LIN {X 0,Y 401.236,Z 607.436,A -85,B 0,C 180,E1 -18756.409,E2 -18756.409} C_VEL
LIN {X 0,Y 401.176,Z 607.446,A -85,B 0,C 180,E1 -18759.805,E2 -18759.805} C_VEL
LIN {X 0,Y 401.178,Z 607.441,A -85,B 0,C 180,E1 -18762.916,E2 -18762.916} C_VEL
LIN {X 0,Y 401.243,Z 607.437,A -85,B 0,C 180,E1 -18765.711,E2 -18765.711} C_VEL
LIN {X 0,Y 401.184,Z 607.441,A -85,B 0,C 180,E1 -18768.656,E2 -18768.656} C_VEL
LIN {X 0,Y 401.211,Z 607.44,A -85,B 0,C 180,E1 -18772.335,E2 -18772.335} C_VEL
LIN {X 0,Y 401.205,Z 607.445,A -85,B 0,C 180,E1 -18776.036,E2 -18776.036} C_VEL
LIN {X 0,Y 401.214,Z 607.439,A -85,B 0,C 180,E1 -18779.583,E2 -18779.583} C_VEL
LIN {X 0,Y 401.241,Z 607.433,A -85,B 0,C 180,E1 -18783.007,E2 -18783.007} C_VEL
LIN {X 0,Y 401.328,Z 607.551,A -85,B 0,C 180,E1 -18783.748,E2 -18783.748} C_VEL
LIN {X 0,Y 403.625,Z 620.57,A -85,B 0,C 180,E1 -18786.89,E2 -18786.89} C_VEL
LIN {X 0,Y 403.581,Z 624.602,A -85,B 0,C 180,E1 -18787.822,E2 -18787.822} C_VEL
LIN {X 0,Y 402.02,Z 640.648,A -85,B 0,C 180,E1 -18791.46,E2 -18791.46} C_VEL
LIN {X 0,Y 401.655,Z 644.543,A -85,B 0,C 180,E1 -18792.313,E2 -18792.313} C_VEL
LIN {X 0,Y 404.651,Z 676.358,A -85,B 0,C 180,E1 -18793.161,E2 -18793.161} C_VEL
LIN {X 0,Y 405.065,Z 683.005,A -85,B 0,C 180,E1 -18793.331,E2 -18793.331} C_VEL
LIN {X 0,Y 403.56,Z 750.603,A -85,B 0,C 180,E1 -18794.942,E2 -18794.942} C_VEL
LIN {X 0,Y 403.184,Z 761.472,A -85,B 0,C 180,E1 -18795.313,E2 -18795.313} C_VEL
LIN {X 0,Y 402.795,Z 771.537,A -85,B 0,C 180,E1 -18795.781,E2 -18795.781} C_VEL
LIN {X 0,Y 402.347,Z 782.009,A -85,B 0,C 180,E1 -18796.407,E2 -18796.407} C_VEL
LIN {X 0,Y 401.883,Z 790.591,A -85,B 0,C 180,E1 -18797.033,E2 -18797.033} C_VEL
LIN {X 0,Y 401.239,Z 800.472,A -85,B 0,C 180,E1 -18797.908,E2 -18797.908} C_VEL
LIN {X 0,Y 400.952,Z 807.903,A -85,B 0,C 180,E1 -18798.679,E2 -18798.679} C_VEL
LIN {X 0,Y 400.256,Z 817.734,A -85,B 0,C 180,E1 -18799.922,E2 -18799.922} C_VEL
LIN {X 0,Y 399.876,Z 824.495,A -85,B 0,C 180,E1 -18800.93,E2 -18800.93} C_VEL
LIN {X 0,Y 399.455,Z 831.571,A -85,B 0,C 180,E1 -18802.19,E2 -18802.19} C_VEL
LIN {X 0,Y 399.275,Z 837.486,A -85,B 0,C 180,E1 -18803.453,E2 -18803.453} C_VEL
LIN {X 0,Y 399.089,Z 843.17,A -85,B 0,C 180,E1 -18804.966,E2 -18804.966} C_VEL
LIN {X 0,Y 399.008,Z 847.589,A -85,B 0,C 180,E1 -18806.478,E2 -18806.478} C_VEL
LIN {X 0,Y 398.99,Z 850.871,A -85,B 0,C 180,E1 -18807.988,E2 -18807.988} C_VEL
LIN {X 0,Y 398.984,Z 852.53,A -85,B 0,C 180,E1 -18808.994,E2 -18808.994} C_VEL
LIN {X 0,Y 398.913,Z 854.339,A -85,B 0,C 180,E1 -18811.006,E2 -18811.006} C_VEL
LIN {X 0,Y 398.916,Z 854.625,A -85,B 0,C 180,E1 -18812.013,E2 -18812.013} C_VEL
LIN {X 0,Y 398.936,Z 853.919,A -85,B 0,C 180,E1 -18814.027,E2 -18814.027} C_VEL
LIN {X 0,Y 399.279,Z 851.395,A -85,B 0,C 180,E1 -18816.042,E2 -18816.042} C_VEL
LIN {X 0,Y 399.537,Z 849.602,A -85,B 0,C 180,E1 -18817.049,E2 -18817.049} C_VEL
LIN {X 0,Y 400.122,Z 845.914,A -85,B 0,C 180,E1 -18818.558,E2 -18818.558} C_VEL
LIN {X 0,Y 400.877,Z 841.119,A -85,B 0,C 180,E1 -18820.063,E2 -18820.063} C_VEL
LIN {X 0,Y 402.106,Z 835.034,A -85,B 0,C 180,E1 -18821.556,E2 -18821.556} C_VEL
LIN {X 0,Y 403.485,Z 827.462,A -85,B 0,C 180,E1 -18823.043,E2 -18823.043} C_VEL
LIN {X 0,Y 404.619,Z 820.376,A -85,B 0,C 180,E1 -18824.204,E2 -18824.204} C_VEL
LIN {X 0,Y 406.142,Z 811.671,A -85,B 0,C 180,E1 -18825.377,E2 -18825.377} C_VEL
LIN {X 0,Y 407.485,Z 803.092,A -85,B 0,C 180,E1 -18826.349,E2 -18826.349} C_VEL
LIN {X 0,Y 408.792,Z 794.302,A -85,B 0,C 180,E1 -18827.192,E2 -18827.192} C_VEL
LIN {X 0,Y 410.234,Z 783.638,A -85,B 0,C 180,E1 -18828.028,E2 -18828.028} C_VEL
LIN {X 0,Y 411.505,Z 773.302,A -85,B 0,C 180,E1 -18828.676,E2 -18828.676} C_VEL
LIN {X 0,Y 412.645,Z 762.627,A -85,B 0,C 180,E1 -18829.201,E2 -18829.201} C_VEL
LIN {X 0,Y 413.498,Z 751.718,A -85,B 0,C 180,E1 -18829.61,E2 -18829.61} C_VEL
LIN {X 0,Y 415.326,Z 717.984,A -85,B 0,C 180,E1 -18830.484,E2 -18830.484} C_VEL
LIN {X 0,Y 416.908,Z 685.447,A -85,B 0,C 180,E1 -18831.33,E2 -18831.33} C_VEL
LIN {X 0,Y 415.184,Z 672.854,A -85,B 0,C 180,E1 -18831.892,E2 -18831.892} C_VEL
LIN {X 0,Y 411.389,Z 654.895,A -85,B 0,C 180,E1 -18832.847,E2 -18832.847} C_VEL
LIN {X 0,Y 407.995,Z 642.009,A -85,B 0,C 180,E1 -18833.66,E2 -18833.66} C_VEL
LIN {X 0,Y 408.232,Z 638.669,A -85,B 0,C 180,E1 -18834.581,E2 -18834.581} C_VEL
LIN {X 0,Y 406.942,Z 630.553,A -85,B 0,C 180,E1 -18837.137,E2 -18837.137} C_VEL
LIN {X 0,Y 405.56,Z 623.765,A -85,B 0,C 180,E1 -18839.487,E2 -18839.487} C_VEL
LIN {X 0,Y 404.026,Z 617.69,A -85,B 0,C 180,E1 -18841.843,E2 -18841.843} C_VEL
LIN {X 0,Y 402.495,Z 611.781,A -85,B 0,C 180,E1 -18844.417,E2 -18844.417} C_VEL
LIN {X 0,Y 401.245,Z 607.433,A -85,B 0,C 180,E1 -18846.636,E2 -18846.636} C_VEL
LIN {X 0,Y 401.201,Z 607.432,A -85,B 0,C 180,E1 -18849.809,E2 -18849.809} C_VEL
LIN {X 0,Y 401.216,Z 607.436,A -85,B 0,C 180,E1 -18852.912,E2 -18852.912} C_VEL
LIN {X 0,Y 401.249,Z 607.434,A -85,B 0,C 180,E1 -18855.712,E2 -18855.712} C_VEL
LIN {X 0,Y 401.218,Z 607.439,A -85,B 0,C 180,E1 -18858.651,E2 -18858.651} C_VEL
LIN {X 0,Y 401.253,Z 607.437,A -85,B 0,C 180,E1 -18861.771,E2 -18861.771} C_VEL
LIN {X 0,Y 401.255,Z 607.436,A -85,B 0,C 180,E1 -18865.13,E2 -18865.13} C_VEL
LIN {X 0,Y 401.243,Z 607.439,A -85,B 0,C 180,E1 -18868.803,E2 -18868.803} C_VEL
LIN {X 0,Y 401.259,Z 607.435,A -85,B 0,C 180,E1 -18871.88,E2 -18871.88} C_VEL
LIN {X 0,Y 401.272,Z 607.436,A -85,B 0,C 180,E1 -18875.232,E2 -18875.232} C_VEL
LIN {X 0,Y 401.283,Z 607.543,A -85,B 0,C 180,E1 -18876.603,E2 -18876.603} C_VEL
LIN {X 0,Y 403.001,Z 613.819,A -85,B 0,C 180,E1 -18879.811,E2 -18879.811} C_VEL
LIN {X 0,Y 404.416,Z 619.422,A -85,B 0,C 180,E1 -18882.288,E2 -18882.288} C_VEL
LIN {X 0,Y 406.124,Z 627.38,A -85,B 0,C 180,E1 -18885.409,E2 -18885.409} C_VEL
LIN {X 0,Y 406.574,Z 629.868,A -85,B 0,C 180,E1 -18886.249,E2 -18886.249} C_VEL
LIN {X 0,Y 412.813,Z 642.686,A -85,B 0,C 180,E1 -18887.379,E2 -18887.379} C_VEL
LIN {X 0,Y 414.891,Z 649.227,A -85,B 0,C 180,E1 -18887.801,E2 -18887.801} C_VEL
LIN {X 0,Y 417.902,Z 663.56,A -85,B 0,C 180,E1 -18888.553,E2 -18888.553} C_VEL
LIN {X 0,Y 414.716,Z 719.256,A -85,B 0,C 180,E1 -18889.969,E2 -18889.969} C_VEL
LIN {X 0,Y 413.649,Z 739.357,A -85,B 0,C 180,E1 -18890.527,E2 -18890.527} C_VEL
LIN {X 0,Y 412.557,Z 752.584,A -85,B 0,C 180,E1 -18891.087,E2 -18891.087} C_VEL
LIN {X 0,Y 411.542,Z 762.975,A -85,B 0,C 180,E1 -18891.682,E2 -18891.682} C_VEL
LIN {X 0,Y 410.218,Z 774.378,A -85,B 0,C 180,E1 -18892.515,E2 -18892.515} C_VEL
LIN {X 0,Y 409.038,Z 783.376,A -85,B 0,C 180,E1 -18893.318,E2 -18893.318} C_VEL
LIN {X 0,Y 407.647,Z 792.758,A -85,B 0,C 180,E1 -18894.33,E2 -18894.33} C_VEL
LIN {X 0,Y 406.417,Z 800.413,A -85,B 0,C 180,E1 -18895.304,E2 -18895.304} C_VEL
LIN {X 0,Y 404.921,Z 808.487,A -85,B 0,C 180,E1 -18896.529,E2 -18896.529} C_VEL
LIN {X 0,Y 403.576,Z 815.234,A -85,B 0,C 180,E1 -18897.762,E2 -18897.762} C_VEL
LIN {X 0,Y 402.452,Z 820.862,A -85,B 0,C 180,E1 -18899.002,E2 -18899.002} C_VEL
LIN {X 0,Y 401.386,Z 826.302,A -85,B 0,C 180,E1 -18900.5,E2 -18900.5} C_VEL
LIN {X 0,Y 400.433,Z 830.57,A -85,B 0,C 180,E1 -18902.005,E2 -18902.005} C_VEL
LIN {X 0,Y 399.986,Z 833.639,A -85,B 0,C 180,E1 -18903.464,E2 -18903.464} C_VEL
LIN {X 0,Y 399.34,Z 836.196,A -85,B 0,C 180,E1 -18905.342,E2 -18905.342} C_VEL
LIN {X 0,Y 399.176,Z 836.861,A -85,B 0,C 180,E1 -18906.043,E2 -18906.043} C_VEL
LIN {X 0,Y 398.808,Z 837.317,A -85,B 0,C 180,E1 -18908.077,E2 -18908.077} C_VEL
LIN {X 0,Y 398.775,Z 836.922,A -85,B 0,C 180,E1 -18909.095,E2 -18909.095} C_VEL
LIN {X 0,Y 398.83,Z 835.693,A -85,B 0,C 180,E1 -18910.421,E2 -18910.421} C_VEL
LIN {X 0,Y 398.746,Z 833,A -85,B 0,C 180,E1 -18912.168,E2 -18912.168} C_VEL
LIN {X 0,Y 398.994,Z 827.975,A -85,B 0,C 180,E1 -18914.227,E2 -18914.227} C_VEL
LIN {X 0,Y 399.221,Z 822.72,A -85,B 0,C 180,E1 -18915.78,E2 -18915.78} C_VEL
LIN {X 0,Y 399.477,Z 817.276,A -85,B 0,C 180,E1 -18917.079,E2 -18917.079} C_VEL
LIN {X 0,Y 399.836,Z 810.653,A -85,B 0,C 180,E1 -18918.38,E2 -18918.38} C_VEL
LIN {X 0,Y 400.296,Z 802.586,A -85,B 0,C 180,E1 -18919.684,E2 -18919.684} C_VEL
LIN {X 0,Y 400.729,Z 794.881,A -85,B 0,C 180,E1 -18920.729,E2 -18920.729} C_VEL
LIN {X 0,Y 401.198,Z 785.777,A -85,B 0,C 180,E1 -18921.764,E2 -18921.764} C_VEL
LIN {X 0,Y 401.706,Z 777.528,A -85,B 0,C 180,E1 -18922.557,E2 -18922.557} C_VEL
LIN {X 0,Y 402.234,Z 767.766,A -85,B 0,C 180,E1 -18923.338,E2 -18923.338} C_VEL
LIN {X 0,Y 402.762,Z 756.608,A -85,B 0,C 180,E1 -18924.054,E2 -18924.054} C_VEL
LIN {X 0,Y 403.039,Z 746.109,A -85,B 0,C 180,E1 -18924.583,E2 -18924.583} C_VEL
LIN {X 0,Y 403.458,Z 734.818,A -85,B 0,C 180,E1 -18925,E2 -18925} C_VEL
LIN {X 0,Y 404.11,Z 711.349,A -85,B 0,C 180,E1 -18925.58,E2 -18925.58} C_VEL
LIN {X 0,Y 405.406,Z 654.841,A -85,B 0,C 180,E1 -18926.917,E2 -18926.917} C_VEL
LIN {X 0,Y 402.416,Z 630.593,A -85,B 0,C 180,E1 -18927.582,E2 -18927.582} C_VEL
LIN {X 0,Y 402.044,Z 626.481,A -85,B 0,C 180,E1 -18927.712,E2 -18927.712} C_VEL
LIN {X 0,Y 402.802,Z 616.204,A -85,B 0,C 180,E1 -18930.284,E2 -18930.284} C_VEL
LIN {X 0,Y 401.358,Z 607.42,A -85,B 0,C 180,E1 -18932.603,E2 -18932.603} C_VEL
LIN {X 0,Y 401.245,Z 607.435,A -85,B 0,C 180,E1 -18936.407,E2 -18936.407} C_VEL
LIN {X 0,Y 401.219,Z 607.441,A -85,B 0,C 180,E1 -18939.812,E2 -18939.812} C_VEL
LIN {X 0,Y 401.232,Z 607.434,A -85,B 0,C 180,E1 -18942.908,E2 -18942.908} C_VEL
LIN {X 0,Y 401.276,Z 607.433,A -85,B 0,C 180,E1 -18945.716,E2 -18945.716} C_VEL
LIN {X 0,Y 401.209,Z 607.438,A -85,B 0,C 180,E1 -18948.651,E2 -18948.651} C_VEL
LIN {X 0,Y 401.249,Z 607.437,A -85,B 0,C 180,E1 -18951.77,E2 -18951.77} C_VEL
LIN {X 0,Y 401.253,Z 607.432,A -85,B 0,C 180,E1 -18955.129,E2 -18955.129} C_VEL
LIN {X 0,Y 401.237,Z 607.434,A -85,B 0,C 180,E1 -18958.803,E2 -18958.803} C_VEL
LIN {X 0,Y 401.254,Z 607.437,A -85,B 0,C 180,E1 -18961.88,E2 -18961.88} C_VEL
LIN {X 0,Y 401.266,Z 607.43,A -85,B 0,C 180,E1 -18965.232,E2 -18965.232} C_VEL
LIN {X 0,Y 401.249,Z 607.434,A -85,B 0,C 180,E1 -18968.494,E2 -18968.494} C_VEL
LIN {X 0,Y 401.293,Z 607.43,A -85,B 0,C 180,E1 -18971.688,E2 -18971.688} C_VEL
LIN {X 0,Y 401.332,Z 607.422,A -85,B 0,C 180,E1 -18974.823,E2 -18974.823} C_VEL
LIN {X 0,Y 401.433,Z 607.416,A -85,B 0,C 180,E1 -18977.914,E2 -18977.914} C_VEL
LIN {X 0,Y 401.48,Z 607.411,A -85,B 0,C 180,E1 -18981.977,E2 -18981.977} C_VEL
LIN {X 0,Y 401.588,Z 607.39,A -85,B 0,C 180,E1 -18984.997,E2 -18984.997} C_VEL
LIN {X 0,Y 401.466,Z 607.412,A -85,B 0,C 180,E1 -18988,E2 -18988} C_VEL
LIN {X 0,Y 401.576,Z 607.399,A -85,B 0,C 180,E1 -18990,E2 -18990} C_VEL
LIN {X 0,Y 401.579,Z 607.398,A -85,B 0,C 180,E1 -18994.001,E2 -18994.001} C_VEL
LIN {X 0,Y 401.5,Z 607.401,A -85,B 0,C 180,E1 -18997.014,E2 -18997.014} C_VEL
LIN {X 0,Y 401.374,Z 607.423,A -85,B 0,C 180,E1 -19000.05,E2 -19000.05} C_VEL
LIN {X 0,Y 401.371,Z 607.417,A -85,B 0,C 180,E1 -19003.113,E2 -19003.113} C_VEL
LIN {X 0,Y 401.354,Z 607.423,A -85,B 0,C 180,E1 -19006.291,E2 -19006.291} C_VEL
LIN {X 0,Y 401.313,Z 607.426,A -85,B 0,C 180,E1 -19009.525,E2 -19009.525} C_VEL
LIN {X 0,Y 401.267,Z 607.431,A -85,B 0,C 180,E1 -19012.583,E2 -19012.583} C_VEL
LIN {X 0,Y 401.279,Z 607.434,A -85,B 0,C 180,E1 -19015.873,E2 -19015.873} C_VEL
LIN {X 0,Y 401.264,Z 607.431,A -85,B 0,C 180,E1 -19019.259,E2 -19019.259} C_VEL
LIN {X 0,Y 401.269,Z 607.43,A -85,B 0,C 180,E1 -19022.76,E2 -19022.76} C_VEL
LIN {X 0,Y 401.311,Z 607.427,A -85,B 0,C 180,E1 -19026.401,E2 -19026.401} C_VEL
LIN {X 0,Y 401.274,Z 607.429,A -85,B 0,C 180,E1 -19028.932,E2 -19028.932} C_VEL
LIN {X 0,Y 401.23,Z 607.435,A -85,B 0,C 180,E1 -19032.909,E2 -19032.909} C_VEL
LIN {X 0,Y 401.274,Z 607.433,A -85,B 0,C 180,E1 -19035.716,E2 -19035.716} C_VEL
LIN {X 0,Y 401.234,Z 607.438,A -85,B 0,C 180,E1 -19039.766,E2 -19039.766} C_VEL
LIN {X 0,Y 401.256,Z 607.434,A -85,B 0,C 180,E1 -19042.341,E2 -19042.341} C_VEL
LIN {X 0,Y 401.258,Z 607.431,A -85,B 0,C 180,E1 -19045.129,E2 -19045.129} C_VEL
LIN {X 0,Y 401.238,Z 607.434,A -85,B 0,C 180,E1 -19048.803,E2 -19048.803} C_VEL
LIN {X 0,Y 401.255,Z 607.437,A -85,B 0,C 180,E1 -19051.88,E2 -19051.88} C_VEL
LIN {X 0,Y 401.257,Z 607.431,A -85,B 0,C 180,E1 -19055.144,E2 -19055.144} C_VEL
LIN {X 0,Y 400.613,Z 607.519,A -85,B 0,C 180,E1 -19055.982,E2 -19055.982} C_VEL
LIN {X 0,Y 397.749,Z 607.869,A -85,B 0,C 180,E1 -19057.345,E2 -19057.345} C_VEL
LIN {X 0,Y 395.32,Z 608.173,A -85,B 0,C 180,E1 -19058.446,E2 -19058.446} C_VEL
LIN {X 0,Y 394.293,Z 608.299,A -85,B 0,C 180,E1 -19059.297,E2 -19059.297} C_VEL
LIN {X 0,Y 394.219,Z 608.307,A -85,B 0,C 180,E1 -19059.586,E2 -19059.586} C_VEL
LIN {X 0,Y 394.213,Z 608.311,A -85,B 0,C 180,E1 -19062.419,E2 -19062.419} C_VEL
LIN {X 0,Y 394.272,Z 608.304,A -85,B 0,C 180,E1 -19065.599,E2 -19065.599} C_VEL
LIN {X 0,Y 394.354,Z 608.292,A -85,B 0,C 180,E1 -19068.733,E2 -19068.733} C_VEL
LIN {X 0,Y 394.435,Z 608.286,A -85,B 0,C 180,E1 -19071.833,E2 -19071.833} C_VEL
LIN {X 0,Y 394.581,Z 608.268,A -85,B 0,C 180,E1 -19073.886,E2 -19073.886} C_VEL
LIN {X 0,Y 394.533,Z 608.269,A -85,B 0,C 180,E1 -19076.947,E2 -19076.947} C_VEL
LIN {X 0,Y 394.53,Z 608.276,A -85,B 0,C 180,E1 -19080,E2 -19080} C_VEL
LIN {X 0,Y 394.544,Z 608.274,A -85,B 0,C 180,E1 -19084.072,E2 -19084.072} C_VEL
LIN {X 0,Y 394.451,Z 608.279,A -85,B 0,C 180,E1 -19087.141,E2 -19087.141} C_VEL
LIN {X 0,Y 394.328,Z 608.299,A -85,B 0,C 180,E1 -19090.232,E2 -19090.232} C_VEL
LIN {X 0,Y 394.389,Z 608.289,A -85,B 0,C 180,E1 -19092.363,E2 -19092.363} C_VEL
LIN {X 0,Y 394.251,Z 608.305,A -85,B 0,C 180,E1 -19095.456,E2 -19095.456} C_VEL
LIN {X 0,Y 394.209,Z 608.31,A -85,B 0,C 180,E1 -19098.653,E2 -19098.653} C_VEL
LIN {X 0,Y 394.241,Z 608.307,A -85,B 0,C 180,E1 -19102.5,E2 -19102.5} C_VEL
LIN {X 0,Y 394.22,Z 608.311,A -85,B 0,C 180,E1 -19106.372,E2 -19106.372} C_VEL
LIN {X 0,Y 394.186,Z 608.317,A -85,B 0,C 180,E1 -19109.838,E2 -19109.838} C_VEL
LIN {X 0,Y 394.177,Z 608.314,A -85,B 0,C 180,E1 -19113.426,E2 -19113.426} C_VEL
LIN {X 0,Y 394.175,Z 608.319,A -85,B 0,C 180,E1 -19115.903,E2 -19115.903} C_VEL
LIN {X 0,Y 394.147,Z 608.318,A -85,B 0,C 180,E1 -19118.563,E2 -19118.563} C_VEL
LIN {X 0,Y 394.145,Z 608.321,A -85,B 0,C 180,E1 -19121.721,E2 -19121.721} C_VEL
LIN {X 0,Y 394.173,Z 608.314,A -85,B 0,C 180,E1 -19125.3,E2 -19125.3} C_VEL
LIN {X 0,Y 394.129,Z 608.319,A -85,B 0,C 180,E1 -19128.886,E2 -19128.886} C_VEL
LIN {X 0,Y 394.17,Z 608.316,A -85,B 0,C 180,E1 -19131.541,E2 -19131.541} C_VEL
LIN {X 0,Y 394.175,Z 608.314,A -85,B 0,C 180,E1 -19134.827,E2 -19134.827} C_VEL
LIN {X 0,Y 394.157,Z 608.317,A -85,B 0,C 180,E1 -19138.539,E2 -19138.539} C_VEL
LIN {X 0,Y 394.172,Z 608.314,A -85,B 0,C 180,E1 -19141.328,E2 -19141.328} C_VEL
LIN {X 0,Y 394.268,Z 608.316,A -85,B 0,C 180,E1 -19143.632,E2 -19143.632} C_VEL
LIN {X 0,Y 396.49,Z 620.927,A -85,B 0,C 180,E1 -19146.728,E2 -19146.728} C_VEL
LIN {X 0,Y 396.582,Z 624.96,A -85,B 0,C 180,E1 -19147.683,E2 -19147.683} C_VEL
LIN {X 0,Y 394.946,Z 640.997,A -85,B 0,C 180,E1 -19151.384,E2 -19151.384} C_VEL
LIN {X 0,Y 394.641,Z 644.341,A -85,B 0,C 180,E1 -19152.138,E2 -19152.138} C_VEL
LIN {X 0,Y 397.593,Z 676.763,A -85,B 0,C 180,E1 -19153.024,E2 -19153.024} C_VEL
LIN {X 0,Y 398.047,Z 682.837,A -85,B 0,C 180,E1 -19153.184,E2 -19153.184} C_VEL
LIN {X 0,Y 396.514,Z 750.366,A -85,B 0,C 180,E1 -19154.831,E2 -19154.831} C_VEL
LIN {X 0,Y 396.1,Z 760.452,A -85,B 0,C 180,E1 -19155.176,E2 -19155.176} C_VEL
LIN {X 0,Y 395.747,Z 770.729,A -85,B 0,C 180,E1 -19155.653,E2 -19155.653} C_VEL
LIN {X 0,Y 395.289,Z 781.328,A -85,B 0,C 180,E1 -19156.291,E2 -19156.291} C_VEL
LIN {X 0,Y 394.759,Z 791.486,A -85,B 0,C 180,E1 -19157.055,E2 -19157.055} C_VEL
LIN {X 0,Y 394.122,Z 800.703,A -85,B 0,C 180,E1 -19157.899,E2 -19157.899} C_VEL
LIN {X 0,Y 393.691,Z 809.348,A -85,B 0,C 180,E1 -19158.844,E2 -19158.844} C_VEL
LIN {X 0,Y 393.206,Z 816.387,A -85,B 0,C 180,E1 -19159.739,E2 -19159.739} C_VEL
LIN {X 0,Y 392.732,Z 824.788,A -85,B 0,C 180,E1 -19161.022,E2 -19161.022} C_VEL
LIN {X 0,Y 392.372,Z 831.779,A -85,B 0,C 180,E1 -19162.306,E2 -19162.306} C_VEL
LIN {X 0,Y 392.171,Z 837.61,A -85,B 0,C 180,E1 -19163.591,E2 -19163.591} C_VEL
LIN {X 0,Y 392.023,Z 842.442,A -85,B 0,C 180,E1 -19164.875,E2 -19164.875} C_VEL
LIN {X 0,Y 391.931,Z 846.998,A -85,B 0,C 180,E1 -19166.414,E2 -19166.414} C_VEL
LIN {X 0,Y 391.919,Z 850.409,A -85,B 0,C 180,E1 -19167.952,E2 -19167.952} C_VEL
LIN {X 0,Y 391.902,Z 852.07,A -85,B 0,C 180,E1 -19168.976,E2 -19168.976} C_VEL
LIN {X 0,Y 391.816,Z 854.109,A -85,B 0,C 180,E1 -19171.025,E2 -19171.025} C_VEL
LIN {X 0,Y 391.84,Z 854.397,A -85,B 0,C 180,E1 -19172.049,E2 -19172.049} C_VEL
LIN {X 0,Y 391.866,Z 853.876,A -85,B 0,C 180,E1 -19174.1,E2 -19174.1} C_VEL
LIN {X 0,Y 392.216,Z 851.508,A -85,B 0,C 180,E1 -19176.151,E2 -19176.151} C_VEL
LIN {X 0,Y 392.673,Z 848.652,A -85,B 0,C 180,E1 -19177.689,E2 -19177.689} C_VEL
LIN {X 0,Y 393.314,Z 844.741,A -85,B 0,C 180,E1 -19179.223,E2 -19179.223} C_VEL
LIN {X 0,Y 394.309,Z 839.666,A -85,B 0,C 180,E1 -19180.75,E2 -19180.75} C_VEL
LIN {X 0,Y 395.397,Z 834.487,A -85,B 0,C 180,E1 -19182.014,E2 -19182.014} C_VEL
LIN {X 0,Y 396.63,Z 828.273,A -85,B 0,C 180,E1 -19183.272,E2 -19183.272} C_VEL
LIN {X 0,Y 398.007,Z 820.325,A -85,B 0,C 180,E1 -19184.609,E2 -19184.609} C_VEL
LIN {X 0,Y 399.577,Z 811.987,A -85,B 0,C 180,E1 -19185.766,E2 -19185.766} C_VEL
LIN {X 0,Y 401.159,Z 802.368,A -85,B 0,C 180,E1 -19186.875,E2 -19186.875} C_VEL
LIN {X 0,Y 402.585,Z 793.445,A -85,B 0,C 180,E1 -19187.727,E2 -19187.727} C_VEL
LIN {X 0,Y 403.855,Z 784.39,A -85,B 0,C 180,E1 -19188.453,E2 -19188.453} C_VEL
LIN {X 0,Y 405.342,Z 773.165,A -85,B 0,C 180,E1 -19189.167,E2 -19189.167} C_VEL
LIN {X 0,Y 406.511,Z 762.53,A -85,B 0,C 180,E1 -19189.699,E2 -19189.699} C_VEL
LIN {X 0,Y 407.384,Z 751.72,A -85,B 0,C 180,E1 -19190.113,E2 -19190.113} C_VEL
LIN {X 0,Y 411.008,Z 686.615,A -85,B 0,C 180,E1 -19191.852,E2 -19191.852} C_VEL
LIN {X 0,Y 409.088,Z 673.009,A -85,B 0,C 180,E1 -19192.489,E2 -19192.489} C_VEL
LIN {X 0,Y 405.833,Z 657.467,A -85,B 0,C 180,E1 -19193.352,E2 -19193.352} C_VEL
LIN {X 0,Y 402.263,Z 644.418,A -85,B 0,C 180,E1 -19194.217,E2 -19194.217} C_VEL
LIN {X 0,Y 401.546,Z 641.756,A -85,B 0,C 180,E1 -19194.412,E2 -19194.412} C_VEL
LIN {X 0,Y 400.497,Z 634.001,A -85,B 0,C 180,E1 -19196.88,E2 -19196.88} C_VEL
LIN {X 0,Y 399.084,Z 626.744,A -85,B 0,C 180,E1 -19199.435,E2 -19199.435} C_VEL
LIN {X 0,Y 397.365,Z 619.783,A -85,B 0,C 180,E1 -19202.209,E2 -19202.209} C_VEL
LIN {X 0,Y 396.08,Z 614.773,A -85,B 0,C 180,E1 -19204.465,E2 -19204.465} C_VEL
LIN {X 0,Y 394.186,Z 608.306,A -85,B 0,C 180,E1 -19207.931,E2 -19207.931} C_VEL
LIN {X 0,Y 394.157,Z 608.31,A -85,B 0,C 180,E1 -19211.723,E2 -19211.723} C_VEL
LIN {X 0,Y 394.178,Z 608.313,A -85,B 0,C 180,E1 -19215.3,E2 -19215.3} C_VEL
LIN {X 0,Y 394.163,Z 608.317,A -85,B 0,C 180,E1 -19218.89,E2 -19218.89} C_VEL
LIN {X 0,Y 394.218,Z 608.313,A -85,B 0,C 180,E1 -19221.546,E2 -19221.546} C_VEL
LIN {X 0,Y 394.2,Z 608.317,A -85,B 0,C 180,E1 -19225.347,E2 -19225.347} C_VEL
LIN {X 0,Y 394.192,Z 608.318,A -85,B 0,C 180,E1 -19228.982,E2 -19228.982} C_VEL
LIN {X 0,Y 394.202,Z 608.313,A -85,B 0,C 180,E1 -19231.331,E2 -19231.331} C_VEL
LIN {X 0,Y 394.221,Z 608.312,A -85,B 0,C 180,E1 -19234.759,E2 -19234.759} C_VEL
LIN {X 0,Y 394.251,Z 608.535,A -85,B 0,C 180,E1 -19235.357,E2 -19235.357} C_VEL
LIN {X 0,Y 395.949,Z 614.585,A -85,B 0,C 180,E1 -19238.737,E2 -19238.737} C_VEL
LIN {X 0,Y 397.48,Z 620.426,A -85,B 0,C 180,E1 -19241.506,E2 -19241.506} C_VEL
LIN {X 0,Y 399.193,Z 628.44,A -85,B 0,C 180,E1 -19244.81,E2 -19244.81} C_VEL
LIN {X 0,Y 399.596,Z 630.251,A -85,B 0,C 180,E1 -19245.436,E2 -19245.436} C_VEL
LIN {X 0,Y 401.549,Z 634.056,A -85,B 0,C 180,E1 -19245.812,E2 -19245.812} C_VEL
LIN {X 0,Y 407.597,Z 646.378,A -85,B 0,C 180,E1 -19246.944,E2 -19246.944} C_VEL
LIN {X 0,Y 409.257,Z 651.668,A -85,B 0,C 180,E1 -19247.307,E2 -19247.307} C_VEL
LIN {X 0,Y 412.093,Z 665.361,A -85,B 0,C 180,E1 -19248.041,E2 -19248.041} C_VEL
LIN {X 0,Y 407.787,Z 735.469,A -85,B 0,C 180,E1 -19249.891,E2 -19249.891} C_VEL
LIN {X 0,Y 406.947,Z 745.966,A -85,B 0,C 180,E1 -19250.276,E2 -19250.276} C_VEL
LIN {X 0,Y 406.062,Z 755.795,A -85,B 0,C 180,E1 -19250.756,E2 -19250.756} C_VEL
LIN {X 0,Y 405.168,Z 764.696,A -85,B 0,C 180,E1 -19251.299,E2 -19251.299} C_VEL
LIN {X 0,Y 403.952,Z 774.477,A -85,B 0,C 180,E1 -19252.026,E2 -19252.026} C_VEL
LIN {X 0,Y 402.65,Z 783.9,A -85,B 0,C 180,E1 -19252.881,E2 -19252.881} C_VEL
LIN {X 0,Y 401.318,Z 792.736,A -85,B 0,C 180,E1 -19253.847,E2 -19253.847} C_VEL
LIN {X 0,Y 399.786,Z 801.361,A -85,B 0,C 180,E1 -19254.974,E2 -19254.974} C_VEL
LIN {X 0,Y 398.525,Z 807.848,A -85,B 0,C 180,E1 -19255.968,E2 -19255.968} C_VEL
LIN {X 0,Y 397.092,Z 814.694,A -85,B 0,C 180,E1 -19257.219,E2 -19257.219} C_VEL
LIN {X 0,Y 395.834,Z 820.474,A -85,B 0,C 180,E1 -19258.479,E2 -19258.479} C_VEL
LIN {X 0,Y 394.645,Z 826.046,A -85,B 0,C 180,E1 -19260,E2 -19260} C_VEL
LIN {X 0,Y 393.65,Z 830.42,A -85,B 0,C 180,E1 -19261.529,E2 -19261.529} C_VEL
LIN {X 0,Y 393.015,Z 833.685,A -85,B 0,C 180,E1 -19263.065,E2 -19263.065} C_VEL
LIN {X 0,Y 392.654,Z 835.313,A -85,B 0,C 180,E1 -19264.091,E2 -19264.091} C_VEL
LIN {X 0,Y 392.069,Z 837.234,A -85,B 0,C 180,E1 -19266.153,E2 -19266.153} C_VEL
LIN {X 0,Y 391.807,Z 837.52,A -85,B 0,C 180,E1 -19267.189,E2 -19267.189} C_VEL
LIN {X 0,Y 391.683,Z 836.895,A -85,B 0,C 180,E1 -19269.261,E2 -19269.261} C_VEL
LIN {X 0,Y 391.735,Z 835.673,A -85,B 0,C 180,E1 -19270.443,E2 -19270.443} C_VEL
LIN {X 0,Y 391.66,Z 832.499,A -85,B 0,C 180,E1 -19272.392,E2 -19272.392} C_VEL
LIN {X 0,Y 391.873,Z 828.652,A -85,B 0,C 180,E1 -19273.963,E2 -19273.963} C_VEL
LIN {X 0,Y 392.105,Z 823.523,A -85,B 0,C 180,E1 -19275.542,E2 -19275.542} C_VEL
LIN {X 0,Y 392.418,Z 816.949,A -85,B 0,C 180,E1 -19277.128,E2 -19277.128} C_VEL
LIN {X 0,Y 392.753,Z 810.207,A -85,B 0,C 180,E1 -19278.454,E2 -19278.454} C_VEL
LIN {X 0,Y 393.148,Z 803.319,A -85,B 0,C 180,E1 -19279.593,E2 -19279.593} C_VEL
LIN {X 0,Y 393.625,Z 795.294,A -85,B 0,C 180,E1 -19280.711,E2 -19280.711} C_VEL
LIN {X 0,Y 394.115,Z 786.144,A -85,B 0,C 180,E1 -19281.777,E2 -19281.777} C_VEL
LIN {X 0,Y 394.628,Z 777.375,A -85,B 0,C 180,E1 -19282.635,E2 -19282.635} C_VEL
LIN {X 0,Y 395.158,Z 768.495,A -85,B 0,C 180,E1 -19283.366,E2 -19283.366} C_VEL
LIN {X 0,Y 395.619,Z 757.479,A -85,B 0,C 180,E1 -19284.099,E2 -19284.099} C_VEL
LIN {X 0,Y 395.968,Z 746.545,A -85,B 0,C 180,E1 -19284.667,E2 -19284.667} C_VEL
LIN {X 0,Y 396.376,Z 735.486,A -85,B 0,C 180,E1 -19285.094,E2 -19285.094} C_VEL
LIN {X 0,Y 397.07,Z 712.336,A -85,B 0,C 180,E1 -19285.684,E2 -19285.684} C_VEL
LIN {X 0,Y 398.332,Z 655.196,A -85,B 0,C 180,E1 -19287.064,E2 -19287.064} C_VEL
LIN {X 0,Y 395.352,Z 630.486,A -85,B 0,C 180,E1 -19287.754,E2 -19287.754} C_VEL
LIN {X 0,Y 395.01,Z 626.722,A -85,B 0,C 180,E1 -19287.862,E2 -19287.862} C_VEL
LIN {X 0,Y 395.756,Z 617.094,A -85,B 0,C 180,E1 -19290.306,E2 -19290.306} C_VEL
LIN {X 0,Y 394.318,Z 608.296,A -85,B 0,C 180,E1 -19292.653,E2 -19292.653} C_VEL
LIN {X 0,Y 394.186,Z 608.318,A -85,B 0,C 180,E1 -19295.901,E2 -19295.901} C_VEL
LIN {X 0,Y 394.192,Z 608.312,A -85,B 0,C 180,E1 -19298.57,E2 -19298.57} C_VEL
LIN {X 0,Y 394.17,Z 608.318,A -85,B 0,C 180,E1 -19301.725,E2 -19301.725} C_VEL
LIN {X 0,Y 394.205,Z 608.31,A -85,B 0,C 180,E1 -19304.704,E2 -19304.704} C_VEL
LIN {X 0,Y 394.172,Z 608.316,A -85,B 0,C 180,E1 -19307.525,E2 -19307.525} C_VEL
LIN {X 0,Y 394.172,Z 608.318,A -85,B 0,C 180,E1 -19310.229,E2 -19310.229} C_VEL
LIN {X 0,Y 394.183,Z 608.312,A -85,B 0,C 180,E1 -19313.094,E2 -19313.094} C_VEL
LIN {X 0,Y 394.197,Z 608.311,A -85,B 0,C 180,E1 -19315.347,E2 -19315.347} C_VEL
LIN {X 0,Y 394.187,Z 608.312,A -85,B 0,C 180,E1 -19318.981,E2 -19318.981} C_VEL
LIN {X 0,Y 394.197,Z 608.311,A -85,B 0,C 180,E1 -19321.33,E2 -19321.33} C_VEL
LIN {X 0,Y 394.216,Z 608.309,A -85,B 0,C 180,E1 -19324.758,E2 -19324.758} C_VEL
LIN {X 0,Y 394.23,Z 608.313,A -85,B 0,C 180,E1 -19328.092,E2 -19328.092} C_VEL
LIN {X 0,Y 394.246,Z 608.305,A -85,B 0,C 180,E1 -19331.349,E2 -19331.349} C_VEL
LIN {X 0,Y 394.304,Z 608.299,A -85,B 0,C 180,E1 -19334.546,E2 -19334.546} C_VEL
LIN {X 0,Y 394.409,Z 608.288,A -85,B 0,C 180,E1 -19337.695,E2 -19337.695} C_VEL
LIN {X 0,Y 394.426,Z 608.287,A -85,B 0,C 180,E1 -19341.832,E2 -19341.832} C_VEL
LIN {X 0,Y 394.534,Z 608.268,A -85,B 0,C 180,E1 -19344.907,E2 -19344.907} C_VEL
LIN {X 0,Y 394.443,Z 608.287,A -85,B 0,C 180,E1 -19347.964,E2 -19347.964} C_VEL
LIN {X 0,Y 394.529,Z 608.277,A -85,B 0,C 180,E1 -19350,E2 -19350} C_VEL
LIN {X 0,Y 394.548,Z 608.273,A -85,B 0,C 180,E1 -19354.072,E2 -19354.072} C_VEL
LIN {X 0,Y 394.447,Z 608.279,A -85,B 0,C 180,E1 -19357.14,E2 -19357.14} C_VEL
LIN {X 0,Y 394.325,Z 608.299,A -85,B 0,C 180,E1 -19360.232,E2 -19360.232} C_VEL
LIN {X 0,Y 394.387,Z 608.29,A -85,B 0,C 180,E1 -19362.364,E2 -19362.364} C_VEL
LIN {X 0,Y 394.305,Z 608.3,A -85,B 0,C 180,E1 -19366.414,E2 -19366.414} C_VEL
LIN {X 0,Y 394.265,Z 608.306,A -85,B 0,C 180,E1 -19369.728,E2 -19369.728} C_VEL
LIN {X 0,Y 394.205,Z 608.309,A -85,B 0,C 180,E1 -19373.011,E2 -19373.011} C_VEL
LIN {X 0,Y 394.217,Z 608.311,A -85,B 0,C 180,E1 -19376.372,E2 -19376.372} C_VEL
LIN {X 0,Y 394.22,Z 608.313,A -85,B 0,C 180,E1 -19379.835,E2 -19379.835} C_VEL
LIN {X 0,Y 394.235,Z 608.307,A -85,B 0,C 180,E1 -19383.421,E2 -19383.421} C_VEL
LIN {X 0,Y 394.258,Z 608.303,A -85,B 0,C 180,E1 -19386.921,E2 -19386.921} C_VEL
LIN {X 0,Y 394.19,Z 608.316,A -85,B 0,C 180,E1 -19390.176,E2 -19390.176} C_VEL
LIN {X 0,Y 394.217,Z 608.314,A -85,B 0,C 180,E1 -19393.864,E2 -19393.864} C_VEL
LIN {X 0,Y 394.175,Z 608.314,A -85,B 0,C 180,E1 -19396.766,E2 -19396.766} C_VEL
LIN {X 0,Y 394.21,Z 608.313,A -85,B 0,C 180,E1 -19400.234,E2 -19400.234} C_VEL
LIN {X 0,Y 394.203,Z 608.31,A -85,B 0,C 180,E1 -19403.091,E2 -19403.091} C_VEL
LIN {X 0,Y 394.201,Z 608.311,A -85,B 0,C 180,E1 -19405.348,E2 -19405.348} C_VEL
LIN {X 0,Y 394.187,Z 608.312,A -85,B 0,C 180,E1 -19408.982,E2 -19408.982} C_VEL
LIN {X 0,Y 394.198,Z 608.311,A -85,B 0,C 180,E1 -19411.331,E2 -19411.331} C_VEL
LIN {X 0,Y 394.217,Z 608.308,A -85,B 0,C 180,E1 -19414.759,E2 -19414.759} C_VEL
LIN {X 0,Y 394.232,Z 608.312,A -85,B 0,C 180,E1 -19418.093,E2 -19418.093} C_VEL
LIN {X 0,Y 394.219,Z 608.307,A -85,B 0,C 180,E1 -19419.586,E2 -19419.586} C_VEL
LIN {X 0,Y 393.573,Z 608.392,A -85,B 0,C 180,E1 -19420.438,E2 -19420.438} C_VEL
LIN {X 0,Y 390.721,Z 608.749,A -85,B 0,C 180,E1 -19421.823,E2 -19421.823} C_VEL
LIN {X 0,Y 388.307,Z 609.046,A -85,B 0,C 180,E1 -19422.943,E2 -19422.943} C_VEL
LIN {X 0,Y 387.292,Z 609.175,A -85,B 0,C 180,E1 -19423.809,E2 -19423.809} C_VEL
LIN {X 0,Y 387.222,Z 609.182,A -85,B 0,C 180,E1 -19424.102,E2 -19424.102} C_VEL
LIN {X 0,Y 387.325,Z 609.169,A -85,B 0,C 180,E1 -19427.565,E2 -19427.565} C_VEL
LIN {X 0,Y 387.399,Z 609.161,A -85,B 0,C 180,E1 -19431.684,E2 -19431.684} C_VEL
LIN {X 0,Y 387.549,Z 609.143,A -85,B 0,C 180,E1 -19433.775,E2 -19433.775} C_VEL
LIN {X 0,Y 387.5,Z 609.145,A -85,B 0,C 180,E1 -19436.892,E2 -19436.892} C_VEL
LIN {X 0,Y 387.486,Z 609.154,A -85,B 0,C 180,E1 -19440,E2 -19440} C_VEL
LIN {X 0,Y 387.513,Z 609.148,A -85,B 0,C 180,E1 -19444.146,E2 -19444.146} C_VEL
LIN {X 0,Y 387.424,Z 609.155,A -85,B 0,C 180,E1 -19447.271,E2 -19447.271} C_VEL
LIN {X 0,Y 387.279,Z 609.175,A -85,B 0,C 180,E1 -19450.42,E2 -19450.42} C_VEL
LIN {X 0,Y 387.335,Z 609.167,A -85,B 0,C 180,E1 -19452.533,E2 -19452.533} C_VEL
LIN {X 0,Y 387.177,Z 609.187,A -85,B 0,C 180,E1 -19456.499,E2 -19456.499} C_VEL
LIN {X 0,Y 387.139,Z 609.195,A -85,B 0,C 180,E1 -19460.107,E2 -19460.107} C_VEL
LIN {X 0,Y 387.16,Z 609.188,A -85,B 0,C 180,E1 -19463.455,E2 -19463.455} C_VEL
LIN {X 0,Y 387.165,Z 609.19,A -85,B 0,C 180,E1 -19465.735,E2 -19465.735} C_VEL
LIN {X 0,Y 387.165,Z 609.187,A -85,B 0,C 180,E1 -19469.241,E2 -19469.241} C_VEL
LIN {X 0,Y 387.12,Z 609.192,A -85,B 0,C 180,E1 -19472.875,E2 -19472.875} C_VEL
LIN {X 0,Y 387.153,Z 609.19,A -85,B 0,C 180,E1 -19475.497,E2 -19475.497} C_VEL
LIN {X 0,Y 387.1,Z 609.195,A -85,B 0,C 180,E1 -19478.916,E2 -19478.916} C_VEL
LIN {X 0,Y 387.096,Z 609.201,A -85,B 0,C 180,E1 -19482.108,E2 -19482.108} C_VEL
LIN {X 0,Y 387.123,Z 609.192,A -85,B 0,C 180,E1 -19485.118,E2 -19485.118} C_VEL
LIN {X 0,Y 387.088,Z 609.203,A -85,B 0,C 180,E1 -19487.97,E2 -19487.97} C_VEL
LIN {X 0,Y 387.098,Z 609.195,A -85,B 0,C 180,E1 -19491.085,E2 -19491.085} C_VEL
LIN {X 0,Y 387.134,Z 609.192,A -85,B 0,C 180,E1 -19494.507,E2 -19494.507} C_VEL
LIN {X 0,Y 387.126,Z 609.194,A -85,B 0,C 180,E1 -19498.351,E2 -19498.351} C_VEL
LIN {X 0,Y 387.151,Z 609.194,A -85,B 0,C 180,E1 -19501.94,E2 -19501.94} C_VEL
LIN {X 0,Y 387.246,Z 609.209,A -85,B 0,C 180,E1 -19503.55,E2 -19503.55} C_VEL
LIN {X 0,Y 389.606,Z 622.967,A -85,B 0,C 180,E1 -19506.982,E2 -19506.982} C_VEL
LIN {X 0,Y 389.034,Z 629.872,A -85,B 0,C 180,E1 -19508.617,E2 -19508.617} C_VEL
LIN {X 0,Y 387.622,Z 644.328,A -85,B 0,C 180,E1 -19511.974,E2 -19511.974} C_VEL
LIN {X 0,Y 390.414,Z 675.899,A -85,B 0,C 180,E1 -19512.845,E2 -19512.845} C_VEL
LIN {X 0,Y 391.068,Z 682.168,A -85,B 0,C 180,E1 -19513.019,E2 -19513.019} C_VEL
LIN {X 0,Y 389.428,Z 750.676,A -85,B 0,C 180,E1 -19514.749,E2 -19514.749} C_VEL
LIN {X 0,Y 389.049,Z 761.325,A -85,B 0,C 180,E1 -19515.134,E2 -19515.134} C_VEL
LIN {X 0,Y 388.639,Z 771.858,A -85,B 0,C 180,E1 -19515.652,E2 -19515.652} C_VEL
LIN {X 0,Y 388.245,Z 780.327,A -85,B 0,C 180,E1 -19516.17,E2 -19516.17} C_VEL
LIN {X 0,Y 387.714,Z 790.621,A -85,B 0,C 180,E1 -19516.949,E2 -19516.949} C_VEL
LIN {X 0,Y 387.054,Z 800.347,A -85,B 0,C 180,E1 -19517.849,E2 -19517.849} C_VEL
LIN {X 0,Y 386.635,Z 808.699,A -85,B 0,C 180,E1 -19518.77,E2 -19518.77} C_VEL
LIN {X 0,Y 386.106,Z 816.695,A -85,B 0,C 180,E1 -19519.812,E2 -19519.812} C_VEL
LIN {X 0,Y 385.594,Z 825.016,A -85,B 0,C 180,E1 -19521.118,E2 -19521.118} C_VEL
LIN {X 0,Y 385.284,Z 831.951,A -85,B 0,C 180,E1 -19522.426,E2 -19522.426} C_VEL
LIN {X 0,Y 385.083,Z 837.724,A -85,B 0,C 180,E1 -19523.735,E2 -19523.735} C_VEL
LIN {X 0,Y 384.969,Z 841.675,A -85,B 0,C 180,E1 -19524.781,E2 -19524.781} C_VEL
LIN {X 0,Y 384.871,Z 846.394,A -85,B 0,C 180,E1 -19526.348,E2 -19526.348} C_VEL
LIN {X 0,Y 384.844,Z 849.934,A -85,B 0,C 180,E1 -19527.914,E2 -19527.914} C_VEL
LIN {X 0,Y 384.83,Z 851.609,A -85,B 0,C 180,E1 -19528.957,E2 -19528.957} C_VEL
LIN {X 0,Y 384.741,Z 853.843,A -85,B 0,C 180,E1 -19531.043,E2 -19531.043} C_VEL
LIN {X 0,Y 384.708,Z 854.183,A -85,B 0,C 180,E1 -19533.131,E2 -19533.131} C_VEL
LIN {X 0,Y 384.782,Z 853.787,A -85,B 0,C 180,E1 -19534.176,E2 -19534.176} C_VEL
LIN {X 0,Y 385.165,Z 851.647,A -85,B 0,C 180,E1 -19536.264,E2 -19536.264} C_VEL
LIN {X 0,Y 385.65,Z 848.914,A -85,B 0,C 180,E1 -19537.829,E2 -19537.829} C_VEL
LIN {X 0,Y 386.313,Z 845.129,A -85,B 0,C 180,E1 -19539.392,E2 -19539.392} C_VEL
LIN {X 0,Y 387.373,Z 840.183,A -85,B 0,C 180,E1 -19540.945,E2 -19540.945} C_VEL
LIN {X 0,Y 388.701,Z 833.988,A -85,B 0,C 180,E1 -19542.489,E2 -19542.489} C_VEL
LIN {X 0,Y 390.078,Z 827.456,A -85,B 0,C 180,E1 -19543.822,E2 -19543.822} C_VEL
LIN {X 0,Y 391.453,Z 820.337,A -85,B 0,C 180,E1 -19545.037,E2 -19545.037} C_VEL
LIN {X 0,Y 393.222,Z 811.356,A -85,B 0,C 180,E1 -19546.294,E2 -19546.294} C_VEL
LIN {X 0,Y 394.712,Z 802.839,A -85,B 0,C 180,E1 -19547.292,E2 -19547.292} C_VEL
LIN {X 0,Y 396.198,Z 794.031,A -85,B 0,C 180,E1 -19548.156,E2 -19548.156} C_VEL
LIN {X 0,Y 397.744,Z 783.399,A -85,B 0,C 180,E1 -19549.014,E2 -19549.014} C_VEL
LIN {X 0,Y 399.176,Z 773.217,A -85,B 0,C 180,E1 -19549.675,E2 -19549.675} C_VEL
LIN {X 0,Y 400.492,Z 762.114,A -85,B 0,C 180,E1 -19550.241,E2 -19550.241} C_VEL
LIN {X 0,Y 401.405,Z 751.458,A -85,B 0,C 180,E1 -19550.66,E2 -19550.66} C_VEL
LIN {X 0,Y 403.619,Z 714.768,A -85,B 0,C 180,E1 -19551.663,E2 -19551.663} C_VEL
LIN {X 0,Y 405.178,Z 687.652,A -85,B 0,C 180,E1 -19552.397,E2 -19552.397} C_VEL
LIN {X 0,Y 402.954,Z 672.521,A -85,B 0,C 180,E1 -19553.146,E2 -19553.146} C_VEL
LIN {X 0,Y 399.703,Z 657.401,A -85,B 0,C 180,E1 -19554.051,E2 -19554.051} C_VEL
LIN {X 0,Y 396.797,Z 647.008,A -85,B 0,C 180,E1 -19554.775,E2 -19554.775} C_VEL
LIN {X 0,Y 395.726,Z 644.343,A -85,B 0,C 180,E1 -19555.012,E2 -19555.012} C_VEL
LIN {X 0,Y 394.619,Z 641.536,A -85,B 0,C 180,E1 -19555.271,E2 -19555.271} C_VEL
LIN {X 0,Y 393.554,Z 634.697,A -85,B 0,C 180,E1 -19557.565,E2 -19557.565} C_VEL
LIN {X 0,Y 392.242,Z 628.103,A -85,B 0,C 180,E1 -19560.001,E2 -19560.001} C_VEL
LIN {X 0,Y 390.367,Z 620.578,A -85,B 0,C 180,E1 -19563.179,E2 -19563.179} C_VEL
LIN {X 0,Y 388.886,Z 615.188,A -85,B 0,C 180,E1 -19565.853,E2 -19565.853} C_VEL
LIN {X 0,Y 387.885,Z 611.644,A -85,B 0,C 180,E1 -19567.878,E2 -19567.878} C_VEL
LIN {X 0,Y 387.116,Z 609.186,A -85,B 0,C 180,E1 -19569.629,E2 -19569.629} C_VEL
LIN {X 0,Y 387.125,Z 609.188,A -85,B 0,C 180,E1 -19572.112,E2 -19572.112} C_VEL
LIN {X 0,Y 387.128,Z 609.192,A -85,B 0,C 180,E1 -19575.119,E2 -19575.119} C_VEL
LIN {X 0,Y 387.134,Z 609.197,A -85,B 0,C 180,E1 -19577.976,E2 -19577.976} C_VEL
LIN {X 0,Y 387.143,Z 609.191,A -85,B 0,C 180,E1 -19581.077,E2 -19581.077} C_VEL
LIN {X 0,Y 387.17,Z 609.188,A -85,B 0,C 180,E1 -19584.625,E2 -19584.625} C_VEL
LIN {X 0,Y 387.145,Z 609.191,A -85,B 0,C 180,E1 -19588.353,E2 -19588.353} C_VEL
LIN {X 0,Y 387.17,Z 609.192,A -85,B 0,C 180,E1 -19590.76,E2 -19590.76} C_VEL
LIN {X 0,Y 387.178,Z 609.199,A -85,B 0,C 180,E1 -19593.69,E2 -19593.69} C_VEL
LIN {X 0,Y 388.538,Z 614.13,A -85,B 0,C 180,E1 -19596.841,E2 -19596.841} C_VEL
LIN {X 0,Y 389.716,Z 618.412,A -85,B 0,C 180,E1 -19599.166,E2 -19599.166} C_VEL
LIN {X 0,Y 391.067,Z 623.634,A -85,B 0,C 180,E1 -19601.676,E2 -19601.676} C_VEL
LIN {X 0,Y 392.485,Z 630.417,A -85,B 0,C 180,E1 -19604.517,E2 -19604.517} C_VEL
LIN {X 0,Y 394.386,Z 634.093,A -85,B 0,C 180,E1 -19604.913,E2 -19604.913} C_VEL
LIN {X 0,Y 399.618,Z 644.067,A -85,B 0,C 180,E1 -19605.945,E2 -19605.945} C_VEL
LIN {X 0,Y 403.254,Z 652.218,A -85,B 0,C 180,E1 -19606.658,E2 -19606.658} C_VEL
LIN {X 0,Y 406.262,Z 666.728,A -85,B 0,C 180,E1 -19607.498,E2 -19607.498} C_VEL
LIN {X 0,Y 401.807,Z 736.089,A -85,B 0,C 180,E1 -19609.358,E2 -19609.358} C_VEL
LIN {X 0,Y 400.85,Z 747.123,A -85,B 0,C 180,E1 -19609.777,E2 -19609.777} C_VEL
LIN {X 0,Y 399.88,Z 757.125,A -85,B 0,C 180,E1 -19610.294,E2 -19610.294} C_VEL
LIN {X 0,Y 398.794,Z 766.591,A -85,B 0,C 180,E1 -19610.904,E2 -19610.904} C_VEL
LIN {X 0,Y 397.54,Z 775.969,A -85,B 0,C 180,E1 -19611.642,E2 -19611.642} C_VEL
LIN {X 0,Y 396.201,Z 785.018,A -85,B 0,C 180,E1 -19612.492,E2 -19612.492} C_VEL
LIN {X 0,Y 394.814,Z 793.677,A -85,B 0,C 180,E1 -19613.467,E2 -19613.467} C_VEL
LIN {X 0,Y 393.538,Z 800.658,A -85,B 0,C 180,E1 -19614.382,E2 -19614.382} C_VEL
LIN {X 0,Y 391.862,Z 808.722,A -85,B 0,C 180,E1 -19615.643,E2 -19615.643} C_VEL
LIN {X 0,Y 390.368,Z 815.462,A -85,B 0,C 180,E1 -19616.914,E2 -19616.914} C_VEL
LIN {X 0,Y 389.286,Z 820.129,A -85,B 0,C 180,E1 -19617.937,E2 -19617.937} C_VEL
LIN {X 0,Y 387.963,Z 825.793,A -85,B 0,C 180,E1 -19619.482,E2 -19619.482} C_VEL
LIN {X 0,Y 386.873,Z 830.274,A -85,B 0,C 180,E1 -19621.037,E2 -19621.037} C_VEL
LIN {X 0,Y 386.262,Z 832.619,A -85,B 0,C 180,E1 -19622.078,E2 -19622.078} C_VEL
LIN {X 0,Y 385.561,Z 835.998,A -85,B 0,C 180,E1 -19624.167,E2 -19624.167} C_VEL
LIN {X 0,Y 384.932,Z 837.524,A -85,B 0,C 180,E1 -19626.268,E2 -19626.268} C_VEL
LIN {X 0,Y 384.692,Z 837.774,A -85,B 0,C 180,E1 -19627.322,E2 -19627.322} C_VEL
LIN {X 0,Y 384.603,Z 836.703,A -85,B 0,C 180,E1 -19629.433,E2 -19629.433} C_VEL
LIN {X 0,Y 384.635,Z 835.621,A -85,B 0,C 180,E1 -19630.492,E2 -19630.492} C_VEL
LIN {X 0,Y 384.547,Z 833.003,A -85,B 0,C 180,E1 -19632.091,E2 -19632.091} C_VEL
LIN {X 0,Y 384.726,Z 829.282,A -85,B 0,C 180,E1 -19633.69,E2 -19633.69} C_VEL
LIN {X 0,Y 384.994,Z 824.068,A -85,B 0,C 180,E1 -19635.363,E2 -19635.363} C_VEL
LIN {X 0,Y 385.248,Z 817.875,A -85,B 0,C 180,E1 -19636.912,E2 -19636.912} C_VEL
LIN {X 0,Y 385.615,Z 811.291,A -85,B 0,C 180,E1 -19638.26,E2 -19638.26} C_VEL
LIN {X 0,Y 386.077,Z 803.194,A -85,B 0,C 180,E1 -19639.624,E2 -19639.624} C_VEL
LIN {X 0,Y 386.528,Z 795.662,A -85,B 0,C 180,E1 -19640.693,E2 -19640.693} C_VEL
LIN {X 0,Y 387.002,Z 786.533,A -85,B 0,C 180,E1 -19641.779,E2 -19641.779} C_VEL
LIN {X 0,Y 387.581,Z 776.958,A -85,B 0,C 180,E1 -19642.726,E2 -19642.726} C_VEL
LIN {X 0,Y 388.135,Z 767.078,A -85,B 0,C 180,E1 -19643.532,E2 -19643.532} C_VEL
LIN {X 0,Y 388.599,Z 756.891,A -85,B 0,C 180,E1 -19644.208,E2 -19644.208} C_VEL
LIN {X 0,Y 388.921,Z 746.508,A -85,B 0,C 180,E1 -19644.754,E2 -19644.754} C_VEL
LIN {X 0,Y 389.323,Z 735.379,A -85,B 0,C 180,E1 -19645.189,E2 -19645.189} C_VEL
LIN {X 0,Y 390.049,Z 710.258,A -85,B 0,C 180,E1 -19645.844,E2 -19645.844} C_VEL
LIN {X 0,Y 391.275,Z 655.609,A -85,B 0,C 180,E1 -19647.212,E2 -19647.212} C_VEL
LIN {X 0,Y 388.182,Z 629.142,A -85,B 0,C 180,E1 -19647.96,E2 -19647.96} C_VEL
LIN {X 0,Y 387.987,Z 626.728,A -85,B 0,C 180,E1 -19648.067,E2 -19648.067} C_VEL
LIN {X 0,Y 388.713,Z 618.084,A -85,B 0,C 180,E1 -19650.301,E2 -19650.301} C_VEL
LIN {X 0,Y 387.269,Z 609.174,A -85,B 0,C 180,E1 -19652.733,E2 -19652.733} C_VEL
LIN {X 0,Y 387.149,Z 609.189,A -85,B 0,C 180,E1 -19656.658,E2 -19656.658} C_VEL
LIN {X 0,Y 387.128,Z 609.192,A -85,B 0,C 180,E1 -19659.291,E2 -19659.291} C_VEL
LIN {X 0,Y 387.119,Z 609.198,A -85,B 0,C 180,E1 -19662.111,E2 -19662.111} C_VEL
LIN {X 0,Y 387.156,Z 609.188,A -85,B 0,C 180,E1 -19665.122,E2 -19665.122} C_VEL
LIN {X 0,Y 387.128,Z 609.198,A -85,B 0,C 180,E1 -19667.975,E2 -19667.975} C_VEL
LIN {X 0,Y 387.135,Z 609.19,A -85,B 0,C 180,E1 -19671.077,E2 -19671.077} C_VEL
LIN {X 0,Y 387.168,Z 609.187,A -85,B 0,C 180,E1 -19674.625,E2 -19674.625} C_VEL
LIN {X 0,Y 387.139,Z 609.193,A -85,B 0,C 180,E1 -19678.352,E2 -19678.352} C_VEL
LIN {X 0,Y 387.165,Z 609.187,A -85,B 0,C 180,E1 -19680.759,E2 -19680.759} C_VEL
LIN {X 0,Y 387.163,Z 609.19,A -85,B 0,C 180,E1 -19684.265,E2 -19684.265} C_VEL
LIN {X 0,Y 387.209,Z 609.184,A -85,B 0,C 180,E1 -19687.673,E2 -19687.673} C_VEL
LIN {X 0,Y 387.2,Z 609.182,A -85,B 0,C 180,E1 -19690.997,E2 -19690.997} C_VEL
LIN {X 0,Y 387.261,Z 609.178,A -85,B 0,C 180,E1 -19694.258,E2 -19694.258} C_VEL
LIN {X 0,Y 387.333,Z 609.168,A -85,B 0,C 180,E1 -19697.557,E2 -19697.557} C_VEL
LIN {X 0,Y 387.391,Z 609.162,A -85,B 0,C 180,E1 -19701.683,E2 -19701.683} C_VEL
LIN {X 0,Y 387.483,Z 609.147,A -85,B 0,C 180,E1 -19704.814,E2 -19704.814} C_VEL
LIN {X 0,Y 387.42,Z 609.161,A -85,B 0,C 180,E1 -19707.928,E2 -19707.928} C_VEL
LIN {X 0,Y 387.485,Z 609.154,A -85,B 0,C 180,E1 -19710,E2 -19710} C_VEL
LIN {X 0,Y 387.517,Z 609.148,A -85,B 0,C 180,E1 -19714.146,E2 -19714.146} C_VEL
LIN {X 0,Y 387.42,Z 609.155,A -85,B 0,C 180,E1 -19717.271,E2 -19717.271} C_VEL
LIN {X 0,Y 387.276,Z 609.175,A -85,B 0,C 180,E1 -19720.42,E2 -19720.42} C_VEL
LIN {X 0,Y 387.333,Z 609.167,A -85,B 0,C 180,E1 -19722.533,E2 -19722.533} C_VEL
LIN {X 0,Y 387.261,Z 609.178,A -85,B 0,C 180,E1 -19725.742,E2 -19725.742} C_VEL
LIN {X 0,Y 387.211,Z 609.186,A -85,B 0,C 180,E1 -19729.84,E2 -19729.84} C_VEL
LIN {X 0,Y 387.16,Z 609.188,A -85,B 0,C 180,E1 -19733.454,E2 -19733.454} C_VEL
LIN {X 0,Y 387.161,Z 609.191,A -85,B 0,C 180,E1 -19735.734,E2 -19735.734} C_VEL
LIN {X 0,Y 387.165,Z 609.187,A -85,B 0,C 180,E1 -19739.24,E2 -19739.24} C_VEL
LIN {X 0,Y 387.173,Z 609.185,A -85,B 0,C 180,E1 -19742.87,E2 -19742.87} C_VEL
LIN {X 0,Y 387.21,Z 609.182,A -85,B 0,C 180,E1 -19746.652,E2 -19746.652} C_VEL
LIN {X 0,Y 387.16,Z 609.188,A -85,B 0,C 180,E1 -19749.288,E2 -19749.288} C_VEL
LIN {X 0,Y 387.118,Z 609.198,A -85,B 0,C 180,E1 -19752.112,E2 -19752.112} C_VEL
LIN {X 0,Y 387.155,Z 609.188,A -85,B 0,C 180,E1 -19755.123,E2 -19755.123} C_VEL
LIN {X 0,Y 387.129,Z 609.198,A -85,B 0,C 180,E1 -19757.976,E2 -19757.976} C_VEL
LIN {X 0,Y 387.158,Z 609.187,A -85,B 0,C 180,E1 -19761.073,E2 -19761.073} C_VEL
LIN {X 0,Y 387.178,Z 609.186,A -85,B 0,C 180,E1 -19764.627,E2 -19764.627} C_VEL
LIN {X 0,Y 387.139,Z 609.193,A -85,B 0,C 180,E1 -19768.353,E2 -19768.353} C_VEL
LIN {X 0,Y 387.166,Z 609.187,A -85,B 0,C 180,E1 -19770.76,E2 -19770.76} C_VEL
LIN {X 0,Y 387.164,Z 609.19,A -85,B 0,C 180,E1 -19774.266,E2 -19774.266} C_VEL
LIN {X 0,Y 387.211,Z 609.184,A -85,B 0,C 180,E1 -19777.674,E2 -19777.674} C_VEL
LIN {X 0,Y 387.198,Z 609.182,A -85,B 0,C 180,E1 -19780.997,E2 -19780.997} C_VEL
LIN {X 0,Y 387.222,Z 609.182,A -85,B 0,C 180,E1 -19784.102,E2 -19784.102} C_VEL
LIN {X 0,Y 386.601,Z 609.264,A -85,B 0,C 180,E1 -19784.971,E2 -19784.971} C_VEL
LIN {X 0,Y 383.807,Z 609.614,A -85,B 0,C 180,E1 -19786.383,E2 -19786.383} C_VEL
LIN {X 0,Y 381.404,Z 609.91,A -85,B 0,C 180,E1 -19787.525,E2 -19787.525} C_VEL
LIN {X 0,Y 380.347,Z 610.039,A -85,B 0,C 180,E1 -19788.407,E2 -19788.407} C_VEL
LIN {X 0,Y 380.249,Z 610.049,A -85,B 0,C 180,E1 -19788.706,E2 -19788.706} C_VEL
LIN {X 0,Y 380.413,Z 610.028,A -85,B 0,C 180,E1 -19792.595,E2 -19792.595} C_VEL
LIN {X 0,Y 380.458,Z 610.022,A -85,B 0,C 180,E1 -19794.719,E2 -19794.719} C_VEL
LIN {X 0,Y 380.403,Z 610.035,A -85,B 0,C 180,E1 -19797.89,E2 -19797.89} C_VEL
LIN {X 0,Y 380.369,Z 610.033,A -85,B 0,C 180,E1 -19801.055,E2 -19801.055} C_VEL
LIN {X 0,Y 380.483,Z 610.023,A -85,B 0,C 180,E1 -19804.223,E2 -19804.223} C_VEL
LIN {X 0,Y 380.379,Z 610.033,A -85,B 0,C 180,E1 -19807.406,E2 -19807.406} C_VEL
LIN {X 0,Y 380.233,Z 610.051,A -85,B 0,C 180,E1 -19810.616,E2 -19810.616} C_VEL
LIN {X 0,Y 380.258,Z 610.047,A -85,B 0,C 180,E1 -19812.771,E2 -19812.771} C_VEL
LIN {X 0,Y 380.124,Z 610.065,A -85,B 0,C 180,E1 -19816.627,E2 -19816.627} C_VEL
LIN {X 0,Y 380.109,Z 610.072,A -85,B 0,C 180,E1 -19819.982,E2 -19819.982} C_VEL
LIN {X 0,Y 380.125,Z 610.063,A -85,B 0,C 180,E1 -19822.878,E2 -19822.878} C_VEL
LIN {X 0,Y 380.113,Z 610.069,A -85,B 0,C 180,E1 -19826.248,E2 -19826.248} C_VEL
LIN {X 0,Y 380.111,Z 610.07,A -85,B 0,C 180,E1 -19829.837,E2 -19829.837} C_VEL
LIN {X 0,Y 380.069,Z 610.073,A -85,B 0,C 180,E1 -19833.565,E2 -19833.565} C_VEL
LIN {X 0,Y 380.083,Z 610.074,A -85,B 0,C 180,E1 -19836.137,E2 -19836.137} C_VEL
LIN {X 0,Y 380.072,Z 610.071,A -85,B 0,C 180,E1 -19839.283,E2 -19839.283} C_VEL
LIN {X 0,Y 380.032,Z 610.075,A -85,B 0,C 180,E1 -19842.997,E2 -19842.997} C_VEL
LIN {X 0,Y 380.06,Z 610.078,A -85,B 0,C 180,E1 -19845.953,E2 -19845.953} C_VEL
LIN {X 0,Y 380.056,Z 610.077,A -85,B 0,C 180,E1 -19849.831,E2 -19849.831} C_VEL
LIN {X 0,Y 380.095,Z 610.068,A -85,B 0,C 180,E1 -19852.546,E2 -19852.546} C_VEL
LIN {X 0,Y 380.057,Z 610.079,A -85,B 0,C 180,E1 -19856.032,E2 -19856.032} C_VEL
LIN {X 0,Y 380.057,Z 610.072,A -85,B 0,C 180,E1 -19858.933,E2 -19858.933} C_VEL
LIN {X 0,Y 380.137,Z 610.063,A -85,B 0,C 180,E1 -19862.571,E2 -19862.571} C_VEL
LIN {X 0,Y 380.176,Z 610.079,A -85,B 0,C 180,E1 -19863.462,E2 -19863.462} C_VEL
LIN {X 0,Y 382.485,Z 623.241,A -85,B 0,C 180,E1 -19866.813,E2 -19866.813} C_VEL
LIN {X 0,Y 382.307,Z 627.869,A -85,B 0,C 180,E1 -19867.939,E2 -19867.939} C_VEL
LIN {X 0,Y 380.581,Z 643.978,A -85,B 0,C 180,E1 -19871.794,E2 -19871.794} C_VEL
LIN {X 0,Y 383.122,Z 673.954,A -85,B 0,C 180,E1 -19872.649,E2 -19872.649} C_VEL
LIN {X 0,Y 384.017,Z 682.677,A -85,B 0,C 180,E1 -19872.899,E2 -19872.899} C_VEL
LIN {X 0,Y 382.35,Z 750.721,A -85,B 0,C 180,E1 -19874.664,E2 -19874.664} C_VEL
LIN {X 0,Y 381.967,Z 761.279,A -85,B 0,C 180,E1 -19875.056,E2 -19875.056} C_VEL
LIN {X 0,Y 381.576,Z 771.779,A -85,B 0,C 180,E1 -19875.584,E2 -19875.584} C_VEL
LIN {X 0,Y 381.139,Z 781.133,A -85,B 0,C 180,E1 -19876.178,E2 -19876.178} C_VEL
LIN {X 0,Y 380.605,Z 791.247,A -85,B 0,C 180,E1 -19876.971,E2 -19876.971} C_VEL
LIN {X 0,Y 379.972,Z 799.975,A -85,B 0,C 180,E1 -19877.795,E2 -19877.795} C_VEL
LIN {X 0,Y 379.578,Z 808.05,A -85,B 0,C 180,E1 -19878.693,E2 -19878.693} C_VEL
LIN {X 0,Y 379.007,Z 817.002,A -85,B 0,C 180,E1 -19879.888,E2 -19879.888} C_VEL
LIN {X 0,Y 378.577,Z 823.79,A -85,B 0,C 180,E1 -19880.952,E2 -19880.952} C_VEL
LIN {X 0,Y 378.215,Z 830.905,A -85,B 0,C 180,E1 -19882.284,E2 -19882.284} C_VEL
LIN {X 0,Y 378.027,Z 836.846,A -85,B 0,C 180,E1 -19883.617,E2 -19883.617} C_VEL
LIN {X 0,Y 377.843,Z 842.559,A -85,B 0,C 180,E1 -19885.215,E2 -19885.215} C_VEL
LIN {X 0,Y 377.768,Z 847.011,A -85,B 0,C 180,E1 -19886.811,E2 -19886.811} C_VEL
LIN {X 0,Y 377.762,Z 849.39,A -85,B 0,C 180,E1 -19887.875,E2 -19887.875} C_VEL
LIN {X 0,Y 377.69,Z 852.538,A -85,B 0,C 180,E1 -19890,E2 -19890} C_VEL
LIN {X 0,Y 377.662,Z 853.496,A -85,B 0,C 180,E1 -19891.063,E2 -19891.063} C_VEL
LIN {X 0,Y 377.622,Z 854.074,A -85,B 0,C 180,E1 -19893.19,E2 -19893.19} C_VEL
LIN {X 0,Y 377.688,Z 853.676,A -85,B 0,C 180,E1 -19894.254,E2 -19894.254} C_VEL
LIN {X 0,Y 378.107,Z 851.765,A -85,B 0,C 180,E1 -19896.382,E2 -19896.382} C_VEL
LIN {X 0,Y 378.605,Z 849.139,A -85,B 0,C 180,E1 -19897.976,E2 -19897.976} C_VEL
LIN {X 0,Y 379.316,Z 845.498,A -85,B 0,C 180,E1 -19899.567,E2 -19899.567} C_VEL
LIN {X 0,Y 380.445,Z 840.756,A -85,B 0,C 180,E1 -19901.147,E2 -19901.147} C_VEL
LIN {X 0,Y 382.095,Z 833.571,A -85,B 0,C 180,E1 -19902.977,E2 -19902.977} C_VEL
LIN {X 0,Y 383.553,Z 826.845,A -85,B 0,C 180,E1 -19904.358,E2 -19904.358} C_VEL
LIN {X 0,Y 385.095,Z 819.778,A -85,B 0,C 180,E1 -19905.562,E2 -19905.562} C_VEL
LIN {X 0,Y 386.865,Z 810.723,A -85,B 0,C 180,E1 -19906.84,E2 -19906.84} C_VEL
LIN {X 0,Y 388.488,Z 802.2,A -85,B 0,C 180,E1 -19907.849,E2 -19907.849} C_VEL
LIN {X 0,Y 390.046,Z 793.413,A -85,B 0,C 180,E1 -19908.724,E2 -19908.724} C_VEL
LIN {X 0,Y 391.706,Z 782.799,A -85,B 0,C 180,E1 -19909.59,E2 -19909.59} C_VEL
LIN {X 0,Y 393.207,Z 772.511,A -85,B 0,C 180,E1 -19910.259,E2 -19910.259} C_VEL
LIN {X 0,Y 394.504,Z 761.963,A -85,B 0,C 180,E1 -19910.8,E2 -19910.8} C_VEL
LIN {X 0,Y 395.469,Z 751.339,A -85,B 0,C 180,E1 -19911.222,E2 -19911.222} C_VEL
LIN {X 0,Y 397.717,Z 715.906,A -85,B 0,C 180,E1 -19912.21,E2 -19912.21} C_VEL
LIN {X 0,Y 399.359,Z 688.629,A -85,B 0,C 180,E1 -19912.978,E2 -19912.978} C_VEL
LIN {X 0,Y 397.365,Z 674.64,A -85,B 0,C 180,E1 -19913.702,E2 -19913.702} C_VEL
LIN {X 0,Y 394.275,Z 660.009,A -85,B 0,C 180,E1 -19914.598,E2 -19914.598} C_VEL
LIN {X 0,Y 391.54,Z 649.746,A -85,B 0,C 180,E1 -19915.344,E2 -19915.344} C_VEL
LIN {X 0,Y 388.912,Z 644.405,A -85,B 0,C 180,E1 -19915.905,E2 -19915.905} C_VEL
LIN {X 0,Y 387.595,Z 641.267,A -85,B 0,C 180,E1 -19916.229,E2 -19916.229} C_VEL
LIN {X 0,Y 386.456,Z 634.342,A -85,B 0,C 180,E1 -19918.706,E2 -19918.706} C_VEL
LIN {X 0,Y 385.033,Z 628.013,A -85,B 0,C 180,E1 -19921.239,E2 -19921.239} C_VEL
LIN {X 0,Y 383.582,Z 622.259,A -85,B 0,C 180,E1 -19923.845,E2 -19923.845} C_VEL
LIN {X 0,Y 382.297,Z 617.617,A -85,B 0,C 180,E1 -19926.277,E2 -19926.277} C_VEL
LIN {X 0,Y 381.127,Z 613.735,A -85,B 0,C 180,E1 -19928.672,E2 -19928.672} C_VEL
LIN {X 0,Y 380.058,Z 610.066,A -85,B 0,C 180,E1 -19931.474,E2 -19931.474} C_VEL
LIN {X 0,Y 380.074,Z 610.074,A -85,B 0,C 180,E1 -19934.452,E2 -19934.452} C_VEL
LIN {X 0,Y 380.086,Z 610.071,A -85,B 0,C 180,E1 -19937.489,E2 -19937.489} C_VEL
LIN {X 0,Y 380.093,Z 610.07,A -85,B 0,C 180,E1 -19941.203,E2 -19941.203} C_VEL
LIN {X 0,Y 380.104,Z 610.068,A -85,B 0,C 180,E1 -19944.176,E2 -19944.176} C_VEL
LIN {X 0,Y 380.099,Z 610.07,A -85,B 0,C 180,E1 -19947.696,E2 -19947.696} C_VEL
LIN {X 0,Y 380.137,Z 610.065,A -85,B 0,C 180,E1 -19950.165,E2 -19950.165} C_VEL
LIN {X 0,Y 380.134,Z 610.093,A -85,B 0,C 180,E1 -19951.835,E2 -19951.835} C_VEL
LIN {X 0,Y 381.346,Z 614.311,A -85,B 0,C 180,E1 -19955.01,E2 -19955.01} C_VEL
LIN {X 0,Y 382.97,Z 620.195,A -85,B 0,C 180,E1 -19958.543,E2 -19958.543} C_VEL
LIN {X 0,Y 384.392,Z 625.807,A -85,B 0,C 180,E1 -19961.362,E2 -19961.362} C_VEL
LIN {X 0,Y 385.465,Z 630.829,A -85,B 0,C 180,E1 -19963.541,E2 -19963.541} C_VEL
LIN {X 0,Y 387.705,Z 634.876,A -85,B 0,C 180,E1 -19964.037,E2 -19964.037} C_VEL
LIN {X 0,Y 392.712,Z 644.139,A -85,B 0,C 180,E1 -19965.084,E2 -19965.084} C_VEL
LIN {X 0,Y 397.748,Z 654.801,A -85,B 0,C 180,E1 -19966.112,E2 -19966.112} C_VEL
LIN {X 0,Y 400.582,Z 668.296,A -85,B 0,C 180,E1 -19966.924,E2 -19966.924} C_VEL
LIN {X 0,Y 395.869,Z 736.647,A -85,B 0,C 180,E1 -19968.809,E2 -19968.809} C_VEL
LIN {X 0,Y 394.875,Z 747.578,A -85,B 0,C 180,E1 -19969.233,E2 -19969.233} C_VEL
LIN {X 0,Y 393.847,Z 757.543,A -85,B 0,C 180,E1 -19969.755,E2 -19969.755} C_VEL
LIN {X 0,Y 392.706,Z 766.976,A -85,B 0,C 180,E1 -19970.374,E2 -19970.374} C_VEL
LIN {X 0,Y 391.402,Z 776.324,A -85,B 0,C 180,E1 -19971.121,E2 -19971.121} C_VEL
LIN {X 0,Y 390.062,Z 784.913,A -85,B 0,C 180,E1 -19971.943,E2 -19971.943} C_VEL
LIN {X 0,Y 388.637,Z 793.066,A -85,B 0,C 180,E1 -19972.866,E2 -19972.866} C_VEL
LIN {X 0,Y 386.955,Z 801.652,A -85,B 0,C 180,E1 -19974.025,E2 -19974.025} C_VEL
LIN {X 0,Y 385.525,Z 808.186,A -85,B 0,C 180,E1 -19975.049,E2 -19975.049} C_VEL
LIN {X 0,Y 383.959,Z 815.055,A -85,B 0,C 180,E1 -19976.339,E2 -19976.339} C_VEL
LIN {X 0,Y 382.497,Z 820.828,A -85,B 0,C 180,E1 -19977.638,E2 -19977.638} C_VEL
LIN {X 0,Y 381.325,Z 825.599,A -85,B 0,C 180,E1 -19978.947,E2 -19978.947} C_VEL
LIN {X 0,Y 380.147,Z 830.157,A -85,B 0,C 180,E1 -19980.528,E2 -19980.528} C_VEL
LIN {X 0,Y 379.183,Z 833.609,A -85,B 0,C 180,E1 -19982.117,E2 -19982.117} C_VEL
LIN {X 0,Y 378.845,Z 835.315,A -85,B 0,C 180,E1 -19983.233,E2 -19983.233} C_VEL
LIN {X 0,Y 378.11,Z 837.476,A -85,B 0,C 180,E1 -19985.314,E2 -19985.314} C_VEL
LIN {X 0,Y 377.575,Z 837.841,A -85,B 0,C 180,E1 -19987.461,E2 -19987.461} C_VEL
LIN {X 0,Y 377.532,Z 837.44,A -85,B 0,C 180,E1 -19988.535,E2 -19988.535} C_VEL
LIN {X 0,Y 377.535,Z 835.219,A -85,B 0,C 180,E1 -19990.692,E2 -19990.692} C_VEL
LIN {X 0,Y 377.482,Z 832.344,A -85,B 0,C 180,E1 -19992.321,E2 -19992.321} C_VEL
LIN {X 0,Y 377.689,Z 828.34,A -85,B 0,C 180,E1 -19993.951,E2 -19993.951} C_VEL
LIN {X 0,Y 377.936,Z 823.479,A -85,B 0,C 180,E1 -19995.476,E2 -19995.476} C_VEL
LIN {X 0,Y 378.172,Z 817.54,A -85,B 0,C 180,E1 -19996.96,E2 -19996.96} C_VEL
LIN {X 0,Y 378.548,Z 810.846,A -85,B 0,C 180,E1 -19998.334,E2 -19998.334} C_VEL
LIN {X 0,Y 378.942,Z 804.164,A -85,B 0,C 180,E1 -19999.49,E2 -19999.49} C_VEL
LIN {X 0,Y 379.462,Z 794.932,A -85,B 0,C 180,E1 -20000.813,E2 -20000.813} C_VEL
LIN {X 0,Y 379.907,Z 786.931,A -85,B 0,C 180,E1 -20001.78,E2 -20001.78} C_VEL
LIN {X 0,Y 380.486,Z 777.422,A -85,B 0,C 180,E1 -20002.742,E2 -20002.742} C_VEL
LIN {X 0,Y 380.991,Z 768.354,A -85,B 0,C 180,E1 -20003.51,E2 -20003.51} C_VEL
LIN {X 0,Y 381.493,Z 757.458,A -85,B 0,C 180,E1 -20004.256,E2 -20004.256} C_VEL
LIN {X 0,Y 381.811,Z 747.204,A -85,B 0,C 180,E1 -20004.812,E2 -20004.812} C_VEL
LIN {X 0,Y 382.208,Z 736.314,A -85,B 0,C 180,E1 -20005.255,E2 -20005.255} C_VEL
LIN {X 0,Y 382.854,Z 716.726,A -85,B 0,C 180,E1 -20005.79,E2 -20005.79} C_VEL
LIN {X 0,Y 384.294,Z 656.62,A -85,B 0,C 180,E1 -20007.331,E2 -20007.331} C_VEL
LIN {X 0,Y 381.084,Z 628.604,A -85,B 0,C 180,E1 -20008.146,E2 -20008.146} C_VEL
LIN {X 0,Y 380.967,Z 627.003,A -85,B 0,C 180,E1 -20008.207,E2 -20008.207} C_VEL
LIN {X 0,Y 381.608,Z 617.859,A -85,B 0,C 180,E1 -20010.613,E2 -20010.613} C_VEL
LIN {X 0,Y 380.243,Z 610.049,A -85,B 0,C 180,E1 -20012.798,E2 -20012.798} C_VEL
LIN {X 0,Y 380.094,Z 610.072,A -85,B 0,C 180,E1 -20016.135,E2 -20016.135} C_VEL
LIN {X 0,Y 380.104,Z 610.067,A -85,B 0,C 180,E1 -20019.289,E2 -20019.289} C_VEL
LIN {X 0,Y 380.09,Z 610.068,A -85,B 0,C 180,E1 -20022.988,E2 -20022.988} C_VEL
LIN {X 0,Y 380.117,Z 610.07,A -85,B 0,C 180,E1 -20025.943,E2 -20025.943} C_VEL
LIN {X 0,Y 380.075,Z 610.075,A -85,B 0,C 180,E1 -20029.833,E2 -20029.833} C_VEL
LIN {X 0,Y 380.117,Z 610.066,A -85,B 0,C 180,E1 -20032.548,E2 -20032.548} C_VEL
LIN {X 0,Y 380.104,Z 610.073,A -85,B 0,C 180,E1 -20036.02,E2 -20036.02} C_VEL
LIN {X 0,Y 380.078,Z 610.069,A -85,B 0,C 180,E1 -20038.935,E2 -20038.935} C_VEL
LIN {X 0,Y 380.119,Z 610.069,A -85,B 0,C 180,E1 -20042.188,E2 -20042.188} C_VEL
LIN {X 0,Y 380.133,Z 610.062,A -85,B 0,C 180,E1 -20044.925,E2 -20044.925} C_VEL
LIN {X 0,Y 380.125,Z 610.066,A -85,B 0,C 180,E1 -20048.375,E2 -20048.375} C_VEL
LIN {X 0,Y 380.162,Z 610.06,A -85,B 0,C 180,E1 -20050.631,E2 -20050.631} C_VEL
LIN {X 0,Y 380.222,Z 610.058,A -85,B 0,C 180,E1 -20053.958,E2 -20053.958} C_VEL
LIN {X 0,Y 380.288,Z 610.044,A -85,B 0,C 180,E1 -20057.47,E2 -20057.47} C_VEL
LIN {X 0,Y 380.338,Z 610.039,A -85,B 0,C 180,E1 -20061.528,E2 -20061.528} C_VEL
LIN {X 0,Y 380.434,Z 610.025,A -85,B 0,C 180,E1 -20064.718,E2 -20064.718} C_VEL
LIN {X 0,Y 380.398,Z 610.035,A -85,B 0,C 180,E1 -20067.889,E2 -20067.889} C_VEL
LIN {X 0,Y 380.369,Z 610.033,A -85,B 0,C 180,E1 -20071.055,E2 -20071.055} C_VEL
LIN {X 0,Y 380.487,Z 610.022,A -85,B 0,C 180,E1 -20074.223,E2 -20074.223} C_VEL
LIN {X 0,Y 380.374,Z 610.034,A -85,B 0,C 180,E1 -20077.406,E2 -20077.406} C_VEL
LIN {X 0,Y 380.229,Z 610.052,A -85,B 0,C 180,E1 -20080.615,E2 -20080.615} C_VEL
LIN {X 0,Y 380.262,Z 610.047,A -85,B 0,C 180,E1 -20082.77,E2 -20082.77} C_VEL
LIN {X 0,Y 380.221,Z 610.058,A -85,B 0,C 180,E1 -20086.041,E2 -20086.041} C_VEL
LIN {X 0,Y 380.179,Z 610.064,A -85,B 0,C 180,E1 -20090.013,E2 -20090.013} C_VEL
LIN {X 0,Y 380.119,Z 610.07,A -85,B 0,C 180,E1 -20093.916,E2 -20093.916} C_VEL
LIN {X 0,Y 380.142,Z 610.063,A -85,B 0,C 180,E1 -20097.429,E2 -20097.429} C_VEL
LIN {X 0,Y 380.101,Z 610.066,A -85,B 0,C 180,E1 -20101.063,E2 -20101.063} C_VEL
LIN {X 0,Y 380.143,Z 610.068,A -85,B 0,C 180,E1 -20103.988,E2 -20103.988} C_VEL
LIN {X 0,Y 380.173,Z 610.059,A -85,B 0,C 180,E1 -20107.445,E2 -20107.445} C_VEL
LIN {X 0,Y 380.066,Z 610.071,A -85,B 0,C 180,E1 -20110.922,E2 -20110.922} C_VEL
LIN {X 0,Y 380.116,Z 610.066,A -85,B 0,C 180,E1 -20114.445,E2 -20114.445} C_VEL
LIN {X 0,Y 380.083,Z 610.07,A -85,B 0,C 180,E1 -20117.489,E2 -20117.489} C_VEL
LIN {X 0,Y 380.107,Z 610.066,A -85,B 0,C 180,E1 -20121.206,E2 -20121.206} C_VEL
LIN {X 0,Y 380.114,Z 610.07,A -85,B 0,C 180,E1 -20124.174,E2 -20124.174} C_VEL
LIN {X 0,Y 380.094,Z 610.071,A -85,B 0,C 180,E1 -20127.696,E2 -20127.696} C_VEL
LIN {X 0,Y 380.132,Z 610.068,A -85,B 0,C 180,E1 -20130.165,E2 -20130.165} C_VEL
LIN {X 0,Y 380.112,Z 610.069,A -85,B 0,C 180,E1 -20133.753,E2 -20133.753} C_VEL
LIN {X 0,Y 380.137,Z 610.063,A -85,B 0,C 180,E1 -20137.236,E2 -20137.236} C_VEL
LIN {X 0,Y 380.162,Z 610.06,A -85,B 0,C 180,E1 -20140.632,E2 -20140.632} C_VEL
LIN {X 0,Y 380.176,Z 610.061,A -85,B 0,C 180,E1 -20144.091,E2 -20144.091} C_VEL
LIN {X 0,Y 380.287,Z 610.045,A -85,B 0,C 180,E1 -20147.474,E2 -20147.474} C_VEL
LIN {X 0,Y 380.249,Z 610.049,A -85,B 0,C 180,E1 -20148.706,E2 -20148.706} C_VEL
LIN {X 0,Y 379.555,Z 610.139,A -85,B 0,C 180,E1 -20149.591,E2 -20149.591} C_VEL
LIN {X 0,Y 376.739,Z 610.485,A -85,B 0,C 180,E1 -20151.03,E2 -20151.03} C_VEL
LIN {X 0,Y 374.422,Z 610.778,A -85,B 0,C 180,E1 -20152.194,E2 -20152.194} C_VEL
LIN {X 0,Y 373.491,Z 610.89,A -85,B 0,C 180,E1 -20153.093,E2 -20153.093} C_VEL
LIN {X 0,Y 373.448,Z 610.896,A -85,B 0,C 180,E1 -20153.397,E2 -20153.397} C_VEL
LIN {X 0,Y 373.411,Z 610.9,A -85,B 0,C 180,E1 -20156.774,E2 -20156.774} C_VEL
LIN {X 0,Y 373.405,Z 610.907,A -85,B 0,C 180,E1 -20160,E2 -20160} C_VEL
LIN {X 0,Y 373.408,Z 610.9,A -85,B 0,C 180,E1 -20163.226,E2 -20163.226} C_VEL
LIN {X 0,Y 373.379,Z 610.906,A -85,B 0,C 180,E1 -20166.463,E2 -20166.463} C_VEL
LIN {X 0,Y 373.233,Z 610.926,A -85,B 0,C 180,E1 -20169.724,E2 -20169.724} C_VEL
LIN {X 0,Y 373.232,Z 610.923,A -85,B 0,C 180,E1 -20172.609,E2 -20172.609} C_VEL
LIN {X 0,Y 373.068,Z 610.943,A -85,B 0,C 180,E1 -20176.757,E2 -20176.757} C_VEL
LIN {X 0,Y 373.081,Z 610.945,A -85,B 0,C 180,E1 -20180.161,E2 -20180.161} C_VEL
LIN {X 0,Y 373.077,Z 610.941,A -85,B 0,C 180,E1 -20183.221,E2 -20183.221} C_VEL
LIN {X 0,Y 373.084,Z 610.941,A -85,B 0,C 180,E1 -20186.782,E2 -20186.782} C_VEL
LIN {X 0,Y 373.024,Z 610.95,A -85,B 0,C 180,E1 -20190.464,E2 -20190.464} C_VEL
LIN {X 0,Y 373.038,Z 610.95,A -85,B 0,C 180,E1 -20194.292,E2 -20194.292} C_VEL
LIN {X 0,Y 373.041,Z 610.946,A -85,B 0,C 180,E1 -20196.931,E2 -20196.931} C_VEL
LIN {X 0,Y 373.032,Z 610.95,A -85,B 0,C 180,E1 -20199.674,E2 -20199.674} C_VEL
LIN {X 0,Y 372.991,Z 610.952,A -85,B 0,C 180,E1 -20202.913,E2 -20202.913} C_VEL
LIN {X 0,Y 373.019,Z 610.956,A -85,B 0,C 180,E1 -20205.991,E2 -20205.991} C_VEL
LIN {X 0,Y 372.982,Z 610.953,A -85,B 0,C 180,E1 -20208.907,E2 -20208.907} C_VEL
LIN {X 0,Y 373.012,Z 610.956,A -85,B 0,C 180,E1 -20212.062,E2 -20212.062} C_VEL
LIN {X 0,Y 373.013,Z 610.952,A -85,B 0,C 180,E1 -20214.401,E2 -20214.401} C_VEL
LIN {X 0,Y 372.994,Z 610.955,A -85,B 0,C 180,E1 -20218.277,E2 -20218.277} C_VEL
LIN {X 0,Y 373.05,Z 610.951,A -85,B 0,C 180,E1 -20222.005,E2 -20222.005} C_VEL
LIN {X 0,Y 373.157,Z 611.122,A -85,B 0,C 180,E1 -20223.43,E2 -20223.43} C_VEL
LIN {X 0,Y 375.292,Z 623.291,A -85,B 0,C 180,E1 -20226.581,E2 -20226.581} C_VEL
LIN {X 0,Y 375.388,Z 627.002,A -85,B 0,C 180,E1 -20227.511,E2 -20227.511} C_VEL
LIN {X 0,Y 373.64,Z 642.994,A -85,B 0,C 180,E1 -20231.416,E2 -20231.416} C_VEL
LIN {X 0,Y 373.542,Z 643.798,A -85,B 0,C 180,E1 -20231.612,E2 -20231.612} C_VEL
LIN {X 0,Y 375.442,Z 667.545,A -85,B 0,C 180,E1 -20232.324,E2 -20232.324} C_VEL
LIN {X 0,Y 376.994,Z 683.026,A -85,B 0,C 180,E1 -20232.776,E2 -20232.776} C_VEL
LIN {X 0,Y 375.273,Z 750.736,A -85,B 0,C 180,E1 -20234.575,E2 -20234.575} C_VEL
LIN {X 0,Y 374.885,Z 761.218,A -85,B 0,C 180,E1 -20234.975,E2 -20234.975} C_VEL
LIN {X 0,Y 374.489,Z 771.68,A -85,B 0,C 180,E1 -20235.513,E2 -20235.513} C_VEL
LIN {X 0,Y 374.099,Z 780.113,A -85,B 0,C 180,E1 -20236.051,E2 -20236.051} C_VEL
LIN {X 0,Y 373.576,Z 790.387,A -85,B 0,C 180,E1 -20236.86,E2 -20236.86} C_VEL
LIN {X 0,Y 372.897,Z 799.535,A -85,B 0,C 180,E1 -20237.732,E2 -20237.732} C_VEL
LIN {X 0,Y 372.418,Z 808.43,A -85,B 0,C 180,E1 -20238.748,E2 -20238.748} C_VEL
LIN {X 0,Y 371.886,Z 817.311,A -85,B 0,C 180,E1 -20239.967,E2 -20239.967} C_VEL
LIN {X 0,Y 371.445,Z 824.022,A -85,B 0,C 180,E1 -20241.05,E2 -20241.05} C_VEL
LIN {X 0,Y 371.112,Z 831.055,A -85,B 0,C 180,E1 -20242.408,E2 -20242.408} C_VEL
LIN {X 0,Y 370.922,Z 836.92,A -85,B 0,C 180,E1 -20243.767,E2 -20243.767} C_VEL
LIN {X 0,Y 370.779,Z 841.778,A -85,B 0,C 180,E1 -20245.124,E2 -20245.124} C_VEL
LIN {X 0,Y 370.696,Z 846.363,A -85,B 0,C 180,E1 -20246.751,E2 -20246.751} C_VEL
LIN {X 0,Y 370.701,Z 848.742,A -85,B 0,C 180,E1 -20247.834,E2 -20247.834} C_VEL
LIN {X 0,Y 370.607,Z 852.167,A -85,B 0,C 180,E1 -20250,E2 -20250} C_VEL
LIN {X 0,Y 370.576,Z 853.125,A -85,B 0,C 180,E1 -20251.083,E2 -20251.083} C_VEL
LIN {X 0,Y 370.531,Z 853.933,A -85,B 0,C 180,E1 -20253.251,E2 -20253.251} C_VEL
LIN {X 0,Y 370.769,Z 852.89,A -85,B 0,C 180,E1 -20255.42,E2 -20255.42} C_VEL
LIN {X 0,Y 371.035,Z 851.821,A -85,B 0,C 180,E1 -20256.504,E2 -20256.504} C_VEL
LIN {X 0,Y 371.773,Z 848.279,A -85,B 0,C 180,E1 -20258.669,E2 -20258.669} C_VEL
LIN {X 0,Y 372.689,Z 844.436,A -85,B 0,C 180,E1 -20260.285,E2 -20260.285} C_VEL
LIN {X 0,Y 373.958,Z 839.441,A -85,B 0,C 180,E1 -20261.89,E2 -20261.89} C_VEL
LIN {X 0,Y 375.538,Z 833.15,A -85,B 0,C 180,E1 -20263.483,E2 -20263.483} C_VEL
LIN {X 0,Y 376.988,Z 826.673,A -85,B 0,C 180,E1 -20264.832,E2 -20264.832} C_VEL
LIN {X 0,Y 378.75,Z 819.317,A -85,B 0,C 180,E1 -20266.106,E2 -20266.106} C_VEL
LIN {X 0,Y 380.621,Z 810.319,A -85,B 0,C 180,E1 -20267.4,E2 -20267.4} C_VEL
LIN {X 0,Y 382.319,Z 801.752,A -85,B 0,C 180,E1 -20268.424,E2 -20268.424} C_VEL
LIN {X 0,Y 383.964,Z 792.897,A -85,B 0,C 180,E1 -20269.308,E2 -20269.308} C_VEL
LIN {X 0,Y 385.721,Z 782.193,A -85,B 0,C 180,E1 -20270.184,E2 -20270.184} C_VEL
LIN {X 0,Y 387.273,Z 771.815,A -85,B 0,C 180,E1 -20270.86,E2 -20270.86} C_VEL
LIN {X 0,Y 388.617,Z 761.149,A -85,B 0,C 180,E1 -20271.407,E2 -20271.407} C_VEL
LIN {X 0,Y 389.631,Z 750.556,A -85,B 0,C 180,E1 -20271.833,E2 -20271.833} C_VEL
LIN {X 0,Y 392.881,Z 703.02,A -85,B 0,C 180,E1 -20273.191,E2 -20273.191} C_VEL
LIN {X 0,Y 393.647,Z 689.784,A -85,B 0,C 180,E1 -20273.578,E2 -20273.578} C_VEL
LIN {X 0,Y 391.816,Z 676.641,A -85,B 0,C 180,E1 -20274.278,E2 -20274.278} C_VEL
LIN {X 0,Y 389.07,Z 662.995,A -85,B 0,C 180,E1 -20275.153,E2 -20275.153} C_VEL
LIN {X 0,Y 386.602,Z 653.573,A -85,B 0,C 180,E1 -20275.855,E2 -20275.855} C_VEL
LIN {X 0,Y 382.52,Z 645.163,A -85,B 0,C 180,E1 -20276.784,E2 -20276.784} C_VEL
LIN {X 0,Y 380.553,Z 640.957,A -85,B 0,C 180,E1 -20277.288,E2 -20277.288} C_VEL
LIN {X 0,Y 379.308,Z 634.123,A -85,B 0,C 180,E1 -20279.907,E2 -20279.907} C_VEL
LIN {X 0,Y 377.867,Z 628.126,A -85,B 0,C 180,E1 -20282.518,E2 -20282.518} C_VEL
LIN {X 0,Y 376.512,Z 622.688,A -85,B 0,C 180,E1 -20285.22,E2 -20285.22} C_VEL
LIN {X 0,Y 375.026,Z 617.499,A -85,B 0,C 180,E1 -20288.331,E2 -20288.331} C_VEL
LIN {X 0,Y 373.765,Z 613.376,A -85,B 0,C 180,E1 -20291.443,E2 -20291.443} C_VEL
LIN {X 0,Y 373.03,Z 610.946,A -85,B 0,C 180,E1 -20294.008,E2 -20294.008} C_VEL
LIN {X 0,Y 373.04,Z 610.948,A -85,B 0,C 180,E1 -20297.471,E2 -20297.471} C_VEL
LIN {X 0,Y 373.048,Z 610.948,A -85,B 0,C 180,E1 -20300.339,E2 -20300.339} C_VEL
LIN {X 0,Y 373.069,Z 610.947,A -85,B 0,C 180,E1 -20303.837,E2 -20303.837} C_VEL
LIN {X 0,Y 373.051,Z 610.95,A -85,B 0,C 180,E1 -20307.009,E2 -20307.009} C_VEL
LIN {X 0,Y 373.069,Z 611.142,A -85,B 0,C 180,E1 -20309.54,E2 -20309.54} C_VEL
LIN {X 0,Y 373.891,Z 613.666,A -85,B 0,C 180,E1 -20312.073,E2 -20312.073} C_VEL
LIN {X 0,Y 374.772,Z 616.821,A -85,B 0,C 180,E1 -20314.541,E2 -20314.541} C_VEL
LIN {X 0,Y 376.097,Z 621.509,A -85,B 0,C 180,E1 -20317.555,E2 -20317.555} C_VEL
LIN {X 0,Y 377.486,Z 626.943,A -85,B 0,C 180,E1 -20320.488,E2 -20320.488} C_VEL
LIN {X 0,Y 378.423,Z 631.136,A -85,B 0,C 180,E1 -20322.461,E2 -20322.461} C_VEL
LIN {X 0,Y 380.582,Z 635.058,A -85,B 0,C 180,E1 -20322.981,E2 -20322.981} C_VEL
LIN {X 0,Y 384.508,Z 641.921,A -85,B 0,C 180,E1 -20323.871,E2 -20323.871} C_VEL
LIN {X 0,Y 389.785,Z 652.008,A -85,B 0,C 180,E1 -20325.003,E2 -20325.003} C_VEL
LIN {X 0,Y 392.811,Z 659.051,A -85,B 0,C 180,E1 -20325.676,E2 -20325.676} C_VEL
LIN {X 0,Y 394.9,Z 669.486,A -85,B 0,C 180,E1 -20326.31,E2 -20326.31} C_VEL
LIN {X 0,Y 390.112,Z 735.868,A -85,B 0,C 180,E1 -20328.182,E2 -20328.182} C_VEL
LIN {X 0,Y 389.101,Z 746.849,A -85,B 0,C 180,E1 -20328.612,E2 -20328.612} C_VEL
LIN {X 0,Y 387.985,Z 756.915,A -85,B 0,C 180,E1 -20329.138,E2 -20329.138} C_VEL
LIN {X 0,Y 386.905,Z 765.64,A -85,B 0,C 180,E1 -20329.701,E2 -20329.701} C_VEL
LIN {X 0,Y 385.525,Z 775.272,A -85,B 0,C 180,E1 -20330.457,E2 -20330.457} C_VEL
LIN {X 0,Y 383.991,Z 784.604,A -85,B 0,C 180,E1 -20331.344,E2 -20331.344} C_VEL
LIN {X 0,Y 382.336,Z 793.541,A -85,B 0,C 180,E1 -20332.367,E2 -20332.367} C_VEL
LIN {X 0,Y 380.738,Z 801.382,A -85,B 0,C 180,E1 -20333.435,E2 -20333.435} C_VEL
LIN {X 0,Y 378.912,Z 809.157,A -85,B 0,C 180,E1 -20334.696,E2 -20334.696} C_VEL
LIN {X 0,Y 377.262,Z 815.848,A -85,B 0,C 180,E1 -20336.007,E2 -20336.007} C_VEL
LIN {X 0,Y 375.723,Z 821.511,A -85,B 0,C 180,E1 -20337.328,E2 -20337.328} C_VEL
LIN {X 0,Y 374.247,Z 826.982,A -85,B 0,C 180,E1 -20338.927,E2 -20338.927} C_VEL
LIN {X 0,Y 373.072,Z 831.252,A -85,B 0,C 180,E1 -20340.538,E2 -20340.538} C_VEL
LIN {X 0,Y 372.104,Z 834.443,A -85,B 0,C 180,E1 -20342.157,E2 -20342.157} C_VEL
LIN {X 0,Y 371.767,Z 836.044,A -85,B 0,C 180,E1 -20343.24,E2 -20343.24} C_VEL
LIN {X 0,Y 370.974,Z 837.821,A -85,B 0,C 180,E1 -20345.417,E2 -20345.417} C_VEL
LIN {X 0,Y 370.701,Z 838.1,A -85,B 0,C 180,E1 -20346.509,E2 -20346.509} C_VEL
LIN {X 0,Y 370.424,Z 837.353,A -85,B 0,C 180,E1 -20348.7,E2 -20348.7} C_VEL
LIN {X 0,Y 370.455,Z 835.362,A -85,B 0,C 180,E1 -20350.516,E2 -20350.516} C_VEL
LIN {X 0,Y 370.376,Z 832.847,A -85,B 0,C 180,E1 -20352.006,E2 -20352.006} C_VEL
LIN {X 0,Y 370.553,Z 828.937,A -85,B 0,C 180,E1 -20353.667,E2 -20353.667} C_VEL
LIN {X 0,Y 370.829,Z 823.76,A -85,B 0,C 180,E1 -20355.333,E2 -20355.333} C_VEL
LIN {X 0,Y 371.064,Z 818.389,A -85,B 0,C 180,E1 -20356.73,E2 -20356.73} C_VEL
LIN {X 0,Y 371.372,Z 811.84,A -85,B 0,C 180,E1 -20358.131,E2 -20358.131} C_VEL
LIN {X 0,Y 371.85,Z 803.937,A -85,B 0,C 180,E1 -20359.526,E2 -20359.526} C_VEL
LIN {X 0,Y 372.37,Z 795.271,A -85,B 0,C 180,E1 -20360.796,E2 -20360.796} C_VEL
LIN {X 0,Y 372.812,Z 787.326,A -85,B 0,C 180,E1 -20361.781,E2 -20361.781} C_VEL
LIN {X 0,Y 373.377,Z 777.85,A -85,B 0,C 180,E1 -20362.762,E2 -20362.762} C_VEL
LIN {X 0,Y 373.923,Z 768.713,A -85,B 0,C 180,E1 -20363.553,E2 -20363.553} C_VEL
LIN {X 0,Y 374.392,Z 758.032,A -85,B 0,C 180,E1 -20364.305,E2 -20364.305} C_VEL
LIN {X 0,Y 374.744,Z 747.146,A -85,B 0,C 180,E1 -20364.906,E2 -20364.906} C_VEL
LIN {X 0,Y 375.143,Z 736.189,A -85,B 0,C 180,E1 -20365.358,E2 -20365.358} C_VEL
LIN {X 0,Y 375.797,Z 716.698,A -85,B 0,C 180,E1 -20365.902,E2 -20365.902} C_VEL
LIN {X 0,Y 377.203,Z 656.755,A -85,B 0,C 180,E1 -20367.475,E2 -20367.475} C_VEL
LIN {X 0,Y 374.055,Z 628.981,A -85,B 0,C 180,E1 -20368.3,E2 -20368.3} C_VEL
LIN {X 0,Y 373.94,Z 627.107,A -85,B 0,C 180,E1 -20368.383,E2 -20368.383} C_VEL
LIN {X 0,Y 374.547,Z 618.642,A -85,B 0,C 180,E1 -20370.655,E2 -20370.655} C_VEL
LIN {X 0,Y 373.186,Z 610.928,A -85,B 0,C 180,E1 -20372.848,E2 -20372.848} C_VEL
LIN {X 0,Y 373.052,Z 610.944,A -85,B 0,C 180,E1 -20376.929,E2 -20376.929} C_VEL
LIN {X 0,Y 373.037,Z 610.95,A -85,B 0,C 180,E1 -20379.673,E2 -20379.673} C_VEL
LIN {X 0,Y 373.067,Z 610.943,A -85,B 0,C 180,E1 -20382.925,E2 -20382.925} C_VEL
LIN {X 0,Y 373.094,Z 610.945,A -85,B 0,C 180,E1 -20386.001,E2 -20386.001} C_VEL
LIN {X 0,Y 373.005,Z 610.951,A -85,B 0,C 180,E1 -20388.91,E2 -20388.91} C_VEL
LIN {X 0,Y 373.05,Z 610.951,A -85,B 0,C 180,E1 -20392.054,E2 -20392.054} C_VEL
LIN {X 0,Y 373.063,Z 610.946,A -85,B 0,C 180,E1 -20395.701,E2 -20395.701} C_VEL
LIN {X 0,Y 373.062,Z 610.945,A -85,B 0,C 180,E1 -20399.54,E2 -20399.54} C_VEL
LIN {X 0,Y 373.081,Z 610.941,A -85,B 0,C 180,E1 -20403.218,E2 -20403.218} C_VEL
LIN {X 0,Y 373.085,Z 610.94,A -85,B 0,C 180,E1 -20406.916,E2 -20406.916} C_VEL
LIN {X 0,Y 373.139,Z 610.938,A -85,B 0,C 180,E1 -20410.251,E2 -20410.251} C_VEL
LIN {X 0,Y 373.19,Z 610.93,A -85,B 0,C 180,E1 -20413.648,E2 -20413.648} C_VEL
LIN {X 0,Y 373.233,Z 610.923,A -85,B 0,C 180,E1 -20417.388,E2 -20417.388} C_VEL
LIN {X 0,Y 373.299,Z 610.915,A -85,B 0,C 180,E1 -20421.367,E2 -20421.367} C_VEL
LIN {X 0,Y 373.386,Z 610.903,A -85,B 0,C 180,E1 -20424.618,E2 -20424.618} C_VEL
LIN {X 0,Y 373.408,Z 610.9,A -85,B 0,C 180,E1 -20426.774,E2 -20426.774} C_VEL
LIN {X 0,Y 373.404,Z 610.908,A -85,B 0,C 180,E1 -20430,E2 -20430} C_VEL
LIN {X 0,Y 373.408,Z 610.9,A -85,B 0,C 180,E1 -20433.226,E2 -20433.226} C_VEL
LIN {X 0,Y 373.375,Z 610.906,A -85,B 0,C 180,E1 -20436.463,E2 -20436.463} C_VEL
LIN {X 0,Y 373.229,Z 610.926,A -85,B 0,C 180,E1 -20439.724,E2 -20439.724} C_VEL
LIN {X 0,Y 373.194,Z 610.927,A -85,B 0,C 180,E1 -20443.016,E2 -20443.016} C_VEL
LIN {X 0,Y 373.175,Z 610.929,A -85,B 0,C 180,E1 -20446.813,E2 -20446.813} C_VEL
LIN {X 0,Y 373.138,Z 610.939,A -85,B 0,C 180,E1 -20450.186,E2 -20450.186} C_VEL
LIN {X 0,Y 373.076,Z 610.942,A -85,B 0,C 180,E1 -20453.22,E2 -20453.22} C_VEL
LIN {X 0,Y 373.08,Z 610.941,A -85,B 0,C 180,E1 -20456.781,E2 -20456.781} C_VEL
LIN {X 0,Y 373.071,Z 610.944,A -85,B 0,C 180,E1 -20460.459,E2 -20460.459} C_VEL
LIN {X 0,Y 373.084,Z 610.94,A -85,B 0,C 180,E1 -20462.987,E2 -20462.987} C_VEL
LIN {X 0,Y 373.107,Z 610.938,A -85,B 0,C 180,E1 -20466.923,E2 -20466.923} C_VEL
LIN {X 0,Y 373.077,Z 610.945,A -85,B 0,C 180,E1 -20469.668,E2 -20469.668} C_VEL
LIN {X 0,Y 373.092,Z 610.946,A -85,B 0,C 180,E1 -20473.998,E2 -20473.998} C_VEL
LIN {X 0,Y 373.038,Z 610.948,A -85,B 0,C 180,E1 -20477.472,E2 -20477.472} C_VEL
LIN {X 0,Y 373.078,Z 610.944,A -85,B 0,C 180,E1 -20480.333,E2 -20480.333} C_VEL
LIN {X 0,Y 373.079,Z 610.945,A -85,B 0,C 180,E1 -20483.834,E2 -20483.834} C_VEL
LIN {X 0,Y 373.047,Z 610.945,A -85,B 0,C 180,E1 -20487.009,E2 -20487.009} C_VEL
LIN {X 0,Y 373.05,Z 610.945,A -85,B 0,C 180,E1 -20490.78,E2 -20490.78} C_VEL
LIN {X 0,Y 373.09,Z 610.942,A -85,B 0,C 180,E1 -20494.418,E2 -20494.418} C_VEL
LIN {X 0,Y 373.069,Z 610.949,A -85,B 0,C 180,E1 -20497.945,E2 -20497.945} C_VEL
LIN {X 0,Y 373.14,Z 610.937,A -85,B 0,C 180,E1 -20500.252,E2 -20500.252} C_VEL
LIN {X 0,Y 373.135,Z 610.936,A -85,B 0,C 180,E1 -20503.646,E2 -20503.646} C_VEL
LIN {X 0,Y 373.23,Z 610.924,A -85,B 0,C 180,E1 -20507.392,E2 -20507.392} C_VEL
LIN {X 0,Y 373.305,Z 610.914,A -85,B 0,C 180,E1 -20511.367,E2 -20511.367} C_VEL
LIN {X 0,Y 373.448,Z 610.896,A -85,B 0,C 180,E1 -20513.397,E2 -20513.397} C_VEL
LIN {X 0,Y 372.864,Z 610.974,A -85,B 0,C 180,E1 -20514.297,E2 -20514.297} C_VEL
LIN {X 0,Y 370.015,Z 611.332,A -85,B 0,C 180,E1 -20515.759,E2 -20515.759} C_VEL
LIN {X 0,Y 367.53,Z 611.64,A -85,B 0,C 180,E1 -20516.942,E2 -20516.942} C_VEL
LIN {X 0,Y 366.432,Z 611.775,A -85,B 0,C 180,E1 -20517.858,E2 -20517.858} C_VEL
LIN {X 0,Y 366.329,Z 611.783,A -85,B 0,C 180,E1 -20518.168,E2 -20518.168} C_VEL
LIN {X 0,Y 366.309,Z 611.784,A -85,B 0,C 180,E1 -20521.096,E2 -20521.096} C_VEL
LIN {X 0,Y 366.424,Z 611.773,A -85,B 0,C 180,E1 -20524.386,E2 -20524.386} C_VEL
LIN {X 0,Y 366.276,Z 611.792,A -85,B 0,C 180,E1 -20527.693,E2 -20527.693} C_VEL
LIN {X 0,Y 366.15,Z 611.804,A -85,B 0,C 180,E1 -20531.029,E2 -20531.029} C_VEL
LIN {X 0,Y 366.118,Z 611.808,A -85,B 0,C 180,E1 -20533.273,E2 -20533.273} C_VEL
LIN {X 0,Y 366.03,Z 611.82,A -85,B 0,C 180,E1 -20536.901,E2 -20536.901} C_VEL
LIN {X 0,Y 366.022,Z 611.823,A -85,B 0,C 180,E1 -20540.332,E2 -20540.332} C_VEL
LIN {X 0,Y 366.021,Z 611.823,A -85,B 0,C 180,E1 -20543.695,E2 -20543.695} C_VEL
LIN {X 0,Y 366.022,Z 611.821,A -85,B 0,C 180,E1 -20547.341,E2 -20547.341} C_VEL
LIN {X 0,Y 365.964,Z 611.827,A -85,B 0,C 180,E1 -20551.116,E2 -20551.116} C_VEL
LIN {X 0,Y 365.987,Z 611.825,A -85,B 0,C 180,E1 -20555.041,E2 -20555.041} C_VEL
LIN {X 0,Y 365.969,Z 611.83,A -85,B 0,C 180,E1 -20558.306,E2 -20558.306} C_VEL
LIN {X 0,Y 365.95,Z 611.835,A -85,B 0,C 180,E1 -20562.061,E2 -20562.061} C_VEL
LIN {X 0,Y 365.993,Z 611.824,A -85,B 0,C 180,E1 -20565.082,E2 -20565.082} C_VEL
LIN {X 0,Y 365.951,Z 611.833,A -85,B 0,C 180,E1 -20568.286,E2 -20568.286} C_VEL
LIN {X 0,Y 365.963,Z 611.83,A -85,B 0,C 180,E1 -20571.696,E2 -20571.696} C_VEL
LIN {X 0,Y 365.952,Z 611.829,A -85,B 0,C 180,E1 -20574.956,E2 -20574.956} C_VEL
LIN {X 0,Y 365.951,Z 611.829,A -85,B 0,C 180,E1 -20578.883,E2 -20578.883} C_VEL
LIN {X 0,Y 366.031,Z 611.819,A -85,B 0,C 180,E1 -20582.66,E2 -20582.66} C_VEL
LIN {X 0,Y 366.118,Z 612.004,A -85,B 0,C 180,E1 -20583.359,E2 -20583.359} C_VEL
LIN {X 0,Y 368.349,Z 624.894,A -85,B 0,C 180,E1 -20586.761,E2 -20586.761} C_VEL
LIN {X 0,Y 368.108,Z 629.518,A -85,B 0,C 180,E1 -20587.926,E2 -20587.926} C_VEL
LIN {X 0,Y 366.518,Z 643.705,A -85,B 0,C 180,E1 -20591.459,E2 -20591.459} C_VEL
LIN {X 0,Y 368.348,Z 667.403,A -85,B 0,C 180,E1 -20592.171,E2 -20592.171} C_VEL
LIN {X 0,Y 369.955,Z 683.489,A -85,B 0,C 180,E1 -20592.651,E2 -20592.651} C_VEL
LIN {X 0,Y 368.197,Z 750.735,A -85,B 0,C 180,E1 -20594.483,E2 -20594.483} C_VEL
LIN {X 0,Y 367.804,Z 761.129,A -85,B 0,C 180,E1 -20594.891,E2 -20594.891} C_VEL
LIN {X 0,Y 367.421,Z 771.525,A -85,B 0,C 180,E1 -20595.44,E2 -20595.44} C_VEL
LIN {X 0,Y 366.972,Z 780.816,A -85,B 0,C 180,E1 -20596.056,E2 -20596.056} C_VEL
LIN {X 0,Y 366.46,Z 790.828,A -85,B 0,C 180,E1 -20596.875,E2 -20596.875} C_VEL
LIN {X 0,Y 365.845,Z 799.108,A -85,B 0,C 180,E1 -20597.682,E2 -20597.682} C_VEL
LIN {X 0,Y 365.387,Z 807.651,A -85,B 0,C 180,E1 -20598.668,E2 -20598.668} C_VEL
LIN {X 0,Y 364.866,Z 815.723,A -85,B 0,C 180,E1 -20599.772,E2 -20599.772} C_VEL
LIN {X 0,Y 364.324,Z 824.104,A -85,B 0,C 180,E1 -20601.153,E2 -20601.153} C_VEL
LIN {X 0,Y 364.049,Z 831.106,A -85,B 0,C 180,E1 -20602.538,E2 -20602.538} C_VEL
LIN {X 0,Y 363.818,Z 836.927,A -85,B 0,C 180,E1 -20603.922,E2 -20603.922} C_VEL
LIN {X 0,Y 363.679,Z 842.542,A -85,B 0,C 180,E1 -20605.582,E2 -20605.582} C_VEL
LIN {X 0,Y 363.637,Z 845.669,A -85,B 0,C 180,E1 -20606.687,E2 -20606.687} C_VEL
LIN {X 0,Y 363.603,Z 849.252,A -85,B 0,C 180,E1 -20608.344,E2 -20608.344} C_VEL
LIN {X 0,Y 363.518,Z 851.747,A -85,B 0,C 180,E1 -20610,E2 -20610} C_VEL
LIN {X 0,Y 363.491,Z 853.449,A -85,B 0,C 180,E1 -20612.209,E2 -20612.209} C_VEL
LIN {X 0,Y 363.456,Z 853.72,A -85,B 0,C 180,E1 -20613.315,E2 -20613.315} C_VEL
LIN {X 0,Y 363.698,Z 852.93,A -85,B 0,C 180,E1 -20615.526,E2 -20615.526} C_VEL
LIN {X 0,Y 363.974,Z 851.862,A -85,B 0,C 180,E1 -20616.631,E2 -20616.631} C_VEL
LIN {X 0,Y 364.753,Z 848.591,A -85,B 0,C 180,E1 -20618.837,E2 -20618.837} C_VEL
LIN {X 0,Y 365.725,Z 844.89,A -85,B 0,C 180,E1 -20620.483,E2 -20620.483} C_VEL
LIN {X 0,Y 367.051,Z 840.058,A -85,B 0,C 180,E1 -20622.117,E2 -20622.117} C_VEL
LIN {X 0,Y 368.701,Z 834.012,A -85,B 0,C 180,E1 -20623.738,E2 -20623.738} C_VEL
LIN {X 0,Y 370.536,Z 826.24,A -85,B 0,C 180,E1 -20625.403,E2 -20625.403} C_VEL
LIN {X 0,Y 372.434,Z 818.969,A -85,B 0,C 180,E1 -20626.667,E2 -20626.667} C_VEL
LIN {X 0,Y 374.2,Z 810.933,A -85,B 0,C 180,E1 -20627.85,E2 -20627.85} C_VEL
LIN {X 0,Y 375.964,Z 802.5,A -85,B 0,C 180,E1 -20628.888,E2 -20628.888} C_VEL
LIN {X 0,Y 377.932,Z 792.4,A -85,B 0,C 180,E1 -20629.911,E2 -20629.911} C_VEL
LIN {X 0,Y 379.523,Z 783.49,A -85,B 0,C 180,E1 -20630.669,E2 -20630.669} C_VEL
LIN {X 0,Y 381.291,Z 772.547,A -85,B 0,C 180,E1 -20631.415,E2 -20631.415} C_VEL
LIN {X 0,Y 382.76,Z 761.644,A -85,B 0,C 180,E1 -20631.998,E2 -20631.998} C_VEL
LIN {X 0,Y 383.906,Z 750.387,A -85,B 0,C 180,E1 -20632.458,E2 -20632.458} C_VEL
LIN {X 0,Y 386.821,Z 709.623,A -85,B 0,C 180,E1 -20633.646,E2 -20633.646} C_VEL
LIN {X 0,Y 388.025,Z 690.926,A -85,B 0,C 180,E1 -20634.197,E2 -20634.197} C_VEL
LIN {X 0,Y 386.294,Z 678.125,A -85,B 0,C 180,E1 -20634.917,E2 -20634.917} C_VEL
LIN {X 0,Y 383.632,Z 664.659,A -85,B 0,C 180,E1 -20635.818,E2 -20635.818} C_VEL
LIN {X 0,Y 381.667,Z 657.266,A -85,B 0,C 180,E1 -20636.394,E2 -20636.394} C_VEL
LIN {X 0,Y 377.751,Z 649.157,A -85,B 0,C 180,E1 -20637.339,E2 -20637.339} C_VEL
LIN {X 0,Y 375.679,Z 645.146,A -85,B 0,C 180,E1 -20637.849,E2 -20637.849} C_VEL
LIN {X 0,Y 373.492,Z 640.65,A -85,B 0,C 180,E1 -20638.445,E2 -20638.445} C_VEL
LIN {X 0,Y 372.165,Z 634.097,A -85,B 0,C 180,E1 -20641.17,E2 -20641.17} C_VEL
LIN {X 0,Y 370.473,Z 627.086,A -85,B 0,C 180,E1 -20644.556,E2 -20644.556} C_VEL
LIN {X 0,Y 368.86,Z 621.119,A -85,B 0,C 180,E1 -20648.085,E2 -20648.085} C_VEL
LIN {X 0,Y 367.313,Z 616.23,A -85,B 0,C 180,E1 -20651.952,E2 -20651.952} C_VEL
LIN {X 0,Y 366.417,Z 613.523,A -85,B 0,C 180,E1 -20655.016,E2 -20655.016} C_VEL
LIN {X 0,Y 365.985,Z 611.831,A -85,B 0,C 180,E1 -20658.161,E2 -20658.161} C_VEL
LIN {X 0,Y 366.007,Z 611.828,A -85,B 0,C 180,E1 -20661.688,E2 -20661.688} C_VEL
LIN {X 0,Y 365.999,Z 611.828,A -85,B 0,C 180,E1 -20665.256,E2 -20665.256} C_VEL
LIN {X 0,Y 366.763,Z 614.234,A -85,B 0,C 180,E1 -20669.251,E2 -20669.251} C_VEL
LIN {X 0,Y 367.418,Z 616.375,A -85,B 0,C 180,E1 -20671.536,E2 -20671.536} C_VEL
LIN {X 0,Y 368.268,Z 619.382,A -85,B 0,C 180,E1 -20674.058,E2 -20674.058} C_VEL
LIN {X 0,Y 369.784,Z 624.89,A -85,B 0,C 180,E1 -20677.738,E2 -20677.738} C_VEL
LIN {X 0,Y 371.284,Z 631.004,A -85,B 0,C 180,E1 -20681.056,E2 -20681.056} C_VEL
LIN {X 0,Y 371.446,Z 631.659,A -85,B 0,C 180,E1 -20681.287,E2 -20681.287} C_VEL
LIN {X 0,Y 373.902,Z 635.818,A -85,B 0,C 180,E1 -20681.927,E2 -20681.927} C_VEL
LIN {X 0,Y 379.529,Z 645.354,A -85,B 0,C 180,E1 -20683.268,E2 -20683.268} C_VEL
LIN {X 0,Y 385.593,Z 657.412,A -85,B 0,C 180,E1 -20684.652,E2 -20684.652} C_VEL
LIN {X 0,Y 387.813,Z 662.851,A -85,B 0,C 180,E1 -20685.169,E2 -20685.169} C_VEL
LIN {X 0,Y 389.302,Z 671.404,A -85,B 0,C 180,E1 -20685.704,E2 -20685.704} C_VEL
LIN {X 0,Y 384.332,Z 737.222,A -85,B 0,C 180,E1 -20687.601,E2 -20687.601} C_VEL
LIN {X 0,Y 383.176,Z 748.605,A -85,B 0,C 180,E1 -20688.065,E2 -20688.065} C_VEL
LIN {X 0,Y 381.84,Z 759.872,A -85,B 0,C 180,E1 -20688.694,E2 -20688.694} C_VEL
LIN {X 0,Y 379.965,Z 772.979,A -85,B 0,C 180,E1 -20689.645,E2 -20689.645} C_VEL
LIN {X 0,Y 378.041,Z 783.84,A -85,B 0,C 180,E1 -20690.67,E2 -20690.67} C_VEL
LIN {X 0,Y 376.315,Z 792.894,A -85,B 0,C 180,E1 -20691.706,E2 -20691.706} C_VEL
LIN {X 0,Y 374.498,Z 801.38,A -85,B 0,C 180,E1 -20692.865,E2 -20692.865} C_VEL
LIN {X 0,Y 372.727,Z 808.771,A -85,B 0,C 180,E1 -20694.067,E2 -20694.067} C_VEL
LIN {X 0,Y 370.938,Z 815.584,A -85,B 0,C 180,E1 -20695.397,E2 -20695.397} C_VEL
LIN {X 0,Y 369.311,Z 821.302,A -85,B 0,C 180,E1 -20696.738,E2 -20696.738} C_VEL
LIN {X 0,Y 367.67,Z 826.826,A -85,B 0,C 180,E1 -20698.362,E2 -20698.362} C_VEL
LIN {X 0,Y 366.349,Z 831.178,A -85,B 0,C 180,E1 -20700,E2 -20700} C_VEL
LIN {X 0,Y 365.632,Z 833.51,A -85,B 0,C 180,E1 -20701.097,E2 -20701.097} C_VEL
LIN {X 0,Y 364.641,Z 836.694,A -85,B 0,C 180,E1 -20703.303,E2 -20703.303} C_VEL
LIN {X 0,Y 363.969,Z 837.941,A -85,B 0,C 180,E1 -20705.108,E2 -20705.108} C_VEL
LIN {X 0,Y 363.583,Z 838.31,A -85,B 0,C 180,E1 -20706.637,E2 -20706.637} C_VEL
LIN {X 0,Y 363.317,Z 837.134,A -85,B 0,C 180,E1 -20708.872,E2 -20708.872} C_VEL
LIN {X 0,Y 363.353,Z 835.183,A -85,B 0,C 180,E1 -20710.534,E2 -20710.534} C_VEL
LIN {X 0,Y 363.279,Z 833.326,A -85,B 0,C 180,E1 -20711.68,E2 -20711.68} C_VEL
LIN {X 0,Y 363.405,Z 829.519,A -85,B 0,C 180,E1 -20713.373,E2 -20713.373} C_VEL
LIN {X 0,Y 363.748,Z 823.429,A -85,B 0,C 180,E1 -20715.353,E2 -20715.353} C_VEL
LIN {X 0,Y 363.98,Z 817.935,A -85,B 0,C 180,E1 -20716.777,E2 -20716.777} C_VEL
LIN {X 0,Y 364.298,Z 811.25,A -85,B 0,C 180,E1 -20718.206,E2 -20718.206} C_VEL
LIN {X 0,Y 364.76,Z 804.088,A -85,B 0,C 180,E1 -20719.487,E2 -20719.487} C_VEL
LIN {X 0,Y 365.254,Z 795.423,A -85,B 0,C 180,E1 -20720.779,E2 -20720.779} C_VEL
LIN {X 0,Y 365.713,Z 787.482,A -85,B 0,C 180,E1 -20721.782,E2 -20721.782} C_VEL
LIN {X 0,Y 366.288,Z 778.049,A -85,B 0,C 180,E1 -20722.782,E2 -20722.782} C_VEL
LIN {X 0,Y 366.847,Z 768.316,A -85,B 0,C 180,E1 -20723.638,E2 -20723.638} C_VEL
LIN {X 0,Y 367.373,Z 757.212,A -85,B 0,C 180,E1 -20724.424,E2 -20724.424} C_VEL
LIN {X 0,Y 367.681,Z 746.852,A -85,B 0,C 180,E1 -20725.003,E2 -20725.003} C_VEL
LIN {X 0,Y 368.105,Z 735.901,A -85,B 0,C 180,E1 -20725.462,E2 -20725.462} C_VEL
LIN {X 0,Y 368.865,Z 712.777,A -85,B 0,C 180,E1 -20726.123,E2 -20726.123} C_VEL
LIN {X 0,Y 370.236,Z 657.813,A -85,B 0,C 180,E1 -20727.597,E2 -20727.597} C_VEL
LIN {X 0,Y 367.097,Z 630.068,A -85,B 0,C 180,E1 -20728.44,E2 -20728.44} C_VEL
LIN {X 0,Y 366.92,Z 627.296,A -85,B 0,C 180,E1 -20728.542,E2 -20728.542} C_VEL
LIN {X 0,Y 367.505,Z 619.77,A -85,B 0,C 180,E1 -20730.593,E2 -20730.593} C_VEL
LIN {X 0,Y 366.145,Z 611.805,A -85,B 0,C 180,E1 -20732.877,E2 -20732.877} C_VEL
LIN {X 0,Y 366.007,Z 611.823,A -85,B 0,C 180,E1 -20736.508,E2 -20736.508} C_VEL
LIN {X 0,Y 365.962,Z 611.834,A -85,B 0,C 180,E1 -20740.04,E2 -20740.04} C_VEL
LIN {X 0,Y 366.042,Z 611.82,A -85,B 0,C 180,E1 -20743.541,E2 -20743.541} C_VEL
LIN {X 0,Y 366.038,Z 611.819,A -85,B 0,C 180,E1 -20746.648,E2 -20746.648} C_VEL
LIN {X 0,Y 365.975,Z 611.827,A -85,B 0,C 180,E1 -20750.832,E2 -20750.832} C_VEL
LIN {X 0,Y 366.021,Z 611.823,A -85,B 0,C 180,E1 -20753.613,E2 -20753.613} C_VEL
LIN {X 0,Y 365.967,Z 611.83,A -85,B 0,C 180,E1 -20756.286,E2 -20756.286} C_VEL
LIN {X 0,Y 366.033,Z 611.82,A -85,B 0,C 180,E1 -20759.442,E2 -20759.442} C_VEL
LIN {X 0,Y 366.019,Z 611.821,A -85,B 0,C 180,E1 -20762.659,E2 -20762.659} C_VEL
LIN {X 0,Y 366.019,Z 611.823,A -85,B 0,C 180,E1 -20766.304,E2 -20766.304} C_VEL
LIN {X 0,Y 366.11,Z 611.815,A -85,B 0,C 180,E1 -20769.856,E2 -20769.856} C_VEL
LIN {X 0,Y 366.133,Z 611.807,A -85,B 0,C 180,E1 -20773.324,E2 -20773.324} C_VEL
LIN {X 0,Y 366.198,Z 611.799,A -85,B 0,C 180,E1 -20777.288,E2 -20777.288} C_VEL
LIN {X 0,Y 366.234,Z 611.794,A -85,B 0,C 180,E1 -20781.199,E2 -20781.199} C_VEL
LIN {X 0,Y 366.341,Z 611.781,A -85,B 0,C 180,E1 -20784.514,E2 -20784.514} C_VEL
LIN {X 0,Y 366.368,Z 611.778,A -85,B 0,C 180,E1 -20786.712,E2 -20786.712} C_VEL
LIN {X 0,Y 366.366,Z 611.784,A -85,B 0,C 180,E1 -20790,E2 -20790} C_VEL
LIN {X 0,Y 366.368,Z 611.778,A -85,B 0,C 180,E1 -20793.288,E2 -20793.288} C_VEL
LIN {X 0,Y 366.373,Z 611.781,A -85,B 0,C 180,E1 -20796.205,E2 -20796.205} C_VEL
LIN {X 0,Y 366.19,Z 611.805,A -85,B 0,C 180,E1 -20799.913,E2 -20799.913} C_VEL
LIN {X 0,Y 366.197,Z 611.799,A -85,B 0,C 180,E1 -20802.711,E2 -20802.711} C_VEL
LIN {X 0,Y 366.132,Z 611.807,A -85,B 0,C 180,E1 -20806.676,E2 -20806.676} C_VEL
LIN {X 0,Y 366.073,Z 611.817,A -85,B 0,C 180,E1 -20810.355,E2 -20810.355} C_VEL
LIN {X 0,Y 366.018,Z 611.824,A -85,B 0,C 180,E1 -20813.695,E2 -20813.695} C_VEL
LIN {X 0,Y 366.018,Z 611.821,A -85,B 0,C 180,E1 -20817.341,E2 -20817.341} C_VEL
LIN {X 0,Y 366.002,Z 611.823,A -85,B 0,C 180,E1 -20821.112,E2 -20821.112} C_VEL
LIN {X 0,Y 366.035,Z 611.819,A -85,B 0,C 180,E1 -20824.63,E2 -20824.63} C_VEL
LIN {X 0,Y 366.039,Z 611.822,A -85,B 0,C 180,E1 -20827.759,E2 -20827.759} C_VEL
LIN {X 0,Y 365.997,Z 611.825,A -85,B 0,C 180,E1 -20830.594,E2 -20830.594} C_VEL
LIN {X 0,Y 366.04,Z 611.819,A -85,B 0,C 180,E1 -20833.542,E2 -20833.542} C_VEL
LIN {X 0,Y 366.036,Z 611.819,A -85,B 0,C 180,E1 -20836.649,E2 -20836.649} C_VEL
LIN {X 0,Y 366.017,Z 611.827,A -85,B 0,C 180,E1 -20839.949,E2 -20839.949} C_VEL
LIN {X 0,Y 366.033,Z 611.821,A -85,B 0,C 180,E1 -20843.615,E2 -20843.615} C_VEL
LIN {X 0,Y 365.996,Z 611.825,A -85,B 0,C 180,E1 -20847.36,E2 -20847.36} C_VEL
LIN {X 0,Y 366.004,Z 611.827,A -85,B 0,C 180,E1 -20850.161,E2 -20850.161} C_VEL
LIN {X 0,Y 366.02,Z 611.82,A -85,B 0,C 180,E1 -20852.66,E2 -20852.66} C_VEL
LIN {X 0,Y 366.021,Z 611.824,A -85,B 0,C 180,E1 -20856.305,E2 -20856.305} C_VEL
LIN {X 0,Y 366.111,Z 611.814,A -85,B 0,C 180,E1 -20859.857,E2 -20859.857} C_VEL
LIN {X 0,Y 366.097,Z 611.811,A -85,B 0,C 180,E1 -20863.323,E2 -20863.323} C_VEL
LIN {X 0,Y 366.196,Z 611.799,A -85,B 0,C 180,E1 -20867.292,E2 -20867.292} C_VEL
LIN {X 0,Y 366.239,Z 611.793,A -85,B 0,C 180,E1 -20871.199,E2 -20871.199} C_VEL
LIN {X 0,Y 366.454,Z 611.769,A -85,B 0,C 180,E1 -20873.684,E2 -20873.684} C_VEL
LIN {X 0,Y 366.371,Z 611.778,A -85,B 0,C 180,E1 -20876.712,E2 -20876.712} C_VEL
LIN {X 0,Y 366.329,Z 611.783,A -85,B 0,C 180,E1 -20878.168,E2 -20878.168} C_VEL
LIN {X 0,Y 365.629,Z 611.87,A -85,B 0,C 180,E1 -20879.086,E2 -20879.086} C_VEL
LIN {X 0,Y 362.778,Z 612.225,A -85,B 0,C 180,E1 -20880.579,E2 -20880.579} C_VEL
LIN {X 0,Y 360.396,Z 612.525,A -85,B 0,C 180,E1 -20881.786,E2 -20881.786} C_VEL
LIN {X 0,Y 359.391,Z 612.646,A -85,B 0,C 180,E1 -20882.72,E2 -20882.72} C_VEL
LIN {X 0,Y 359.318,Z 612.654,A -85,B 0,C 180,E1 -20883.036,E2 -20883.036} C_VEL
LIN {X 0,Y 359.33,Z 612.659,A -85,B 0,C 180,E1 -20886.204,E2 -20886.204} C_VEL
LIN {X 0,Y 359.141,Z 612.682,A -85,B 0,C 180,E1 -20890.11,E2 -20890.11} C_VEL
LIN {X 0,Y 359.157,Z 612.675,A -85,B 0,C 180,E1 -20892.807,E2 -20892.807} C_VEL
LIN {X 0,Y 358.986,Z 612.697,A -85,B 0,C 180,E1 -20897.045,E2 -20897.045} C_VEL
LIN {X 0,Y 358.977,Z 612.698,A -85,B 0,C 180,E1 -20900.562,E2 -20900.562} C_VEL
LIN {X 0,Y 358.963,Z 612.704,A -85,B 0,C 180,E1 -20904.191,E2 -20904.191} C_VEL
LIN {X 0,Y 358.958,Z 612.701,A -85,B 0,C 180,E1 -20906.667,E2 -20906.667} C_VEL
LIN {X 0,Y 358.943,Z 612.702,A -85,B 0,C 180,E1 -20909.2,E2 -20909.2} C_VEL
LIN {X 0,Y 358.905,Z 612.706,A -85,B 0,C 180,E1 -20912.945,E2 -20912.945} C_VEL
LIN {X 0,Y 358.948,Z 612.706,A -85,B 0,C 180,E1 -20915.832,E2 -20915.832} C_VEL
LIN {X 0,Y 358.913,Z 612.706,A -85,B 0,C 180,E1 -20918.682,E2 -20918.682} C_VEL
LIN {X 0,Y 358.915,Z 612.71,A -85,B 0,C 180,E1 -20922.133,E2 -20922.133} C_VEL
LIN {X 0,Y 358.931,Z 612.705,A -85,B 0,C 180,E1 -20925.37,E2 -20925.37} C_VEL
LIN {X 0,Y 358.9,Z 612.709,A -85,B 0,C 180,E1 -20928.428,E2 -20928.428} C_VEL
LIN {X 0,Y 358.908,Z 612.706,A -85,B 0,C 180,E1 -20931.354,E2 -20931.354} C_VEL
LIN {X 0,Y 358.911,Z 612.711,A -85,B 0,C 180,E1 -20934.164,E2 -20934.164} C_VEL
LIN {X 0,Y 358.895,Z 612.708,A -85,B 0,C 180,E1 -20937.058,E2 -20937.058} C_VEL
LIN {X 0,Y 358.946,Z 612.703,A -85,B 0,C 180,E1 -20939.512,E2 -20939.512} C_VEL
LIN {X 0,Y 359.063,Z 612.792,A -85,B 0,C 180,E1 -20943.263,E2 -20943.263} C_VEL
LIN {X 0,Y 361.196,Z 625.084,A -85,B 0,C 180,E1 -20946.575,E2 -20946.575} C_VEL
LIN {X 0,Y 361.229,Z 628.584,A -85,B 0,C 180,E1 -20947.483,E2 -20947.483} C_VEL
LIN {X 0,Y 359.483,Z 643.537,A -85,B 0,C 180,E1 -20951.283,E2 -20951.283} C_VEL
LIN {X 0,Y 361.179,Z 666.843,A -85,B 0,C 180,E1 -20952.003,E2 -20952.003} C_VEL
LIN {X 0,Y 362.9,Z 684.343,A -85,B 0,C 180,E1 -20952.536,E2 -20952.536} C_VEL
LIN {X 0,Y 361.16,Z 750.046,A -85,B 0,C 180,E1 -20954.39,E2 -20954.39} C_VEL
LIN {X 0,Y 360.707,Z 760.473,A -85,B 0,C 180,E1 -20954.802,E2 -20954.802} C_VEL
LIN {X 0,Y 360.371,Z 770.995,A -85,B 0,C 180,E1 -20955.364,E2 -20955.364} C_VEL
LIN {X 0,Y 359.866,Z 781.249,A -85,B 0,C 180,E1 -20956.062,E2 -20956.062} C_VEL
LIN {X 0,Y 359.347,Z 791.224,A -85,B 0,C 180,E1 -20956.904,E2 -20956.904} C_VEL
LIN {X 0,Y 358.752,Z 799.101,A -85,B 0,C 180,E1 -20957.692,E2 -20957.692} C_VEL
LIN {X 0,Y 358.257,Z 807.823,A -85,B 0,C 180,E1 -20958.725,E2 -20958.725} C_VEL
LIN {X 0,Y 357.763,Z 815.851,A -85,B 0,C 180,E1 -20959.851,E2 -20959.851} C_VEL
LIN {X 0,Y 357.242,Z 824.191,A -85,B 0,C 180,E1 -20961.26,E2 -20961.26} C_VEL
LIN {X 0,Y 356.96,Z 831.152,A -85,B 0,C 180,E1 -20962.672,E2 -20962.672} C_VEL
LIN {X 0,Y 356.765,Z 835.939,A -85,B 0,C 180,E1 -20963.801,E2 -20963.801} C_VEL
LIN {X 0,Y 356.604,Z 841.729,A -85,B 0,C 180,E1 -20965.494,E2 -20965.494} C_VEL
LIN {X 0,Y 356.555,Z 846.245,A -85,B 0,C 180,E1 -20967.185,E2 -20967.185} C_VEL
LIN {X 0,Y 356.515,Z 849.606,A -85,B 0,C 180,E1 -20968.874,E2 -20968.874} C_VEL
LIN {X 0,Y 356.451,Z 851.245,A -85,B 0,C 180,E1 -20970,E2 -20970} C_VEL
LIN {X 0,Y 356.404,Z 853.201,A -85,B 0,C 180,E1 -20972.253,E2 -20972.253} C_VEL
LIN {X 0,Y 356.454,Z 853.358,A -85,B 0,C 180,E1 -20974.508,E2 -20974.508} C_VEL
LIN {X 0,Y 356.638,Z 852.932,A -85,B 0,C 180,E1 -20975.636,E2 -20975.636} C_VEL
LIN {X 0,Y 357.274,Z 850.572,A -85,B 0,C 180,E1 -20977.888,E2 -20977.888} C_VEL
LIN {X 0,Y 358.088,Z 847.712,A -85,B 0,C 180,E1 -20979.571,E2 -20979.571} C_VEL
LIN {X 0,Y 359.162,Z 843.847,A -85,B 0,C 180,E1 -20981.246,E2 -20981.246} C_VEL
LIN {X 0,Y 360.683,Z 838.833,A -85,B 0,C 180,E1 -20982.905,E2 -20982.905} C_VEL
LIN {X 0,Y 362.501,Z 832.538,A -85,B 0,C 180,E1 -20984.548,E2 -20984.548} C_VEL
LIN {X 0,Y 364.015,Z 826.371,A -85,B 0,C 180,E1 -20985.886,E2 -20985.886} C_VEL
LIN {X 0,Y 366.127,Z 818.62,A -85,B 0,C 180,E1 -20987.25,E2 -20987.25} C_VEL
LIN {X 0,Y 368.005,Z 810.605,A -85,B 0,C 180,E1 -20988.448,E2 -20988.448} C_VEL
LIN {X 0,Y 369.89,Z 802.246,A -85,B 0,C 180,E1 -20989.497,E2 -20989.497} C_VEL
LIN {X 0,Y 371.964,Z 792.237,A -85,B 0,C 180,E1 -20990.532,E2 -20990.532} C_VEL
LIN {X 0,Y 373.666,Z 783.301,A -85,B 0,C 180,E1 -20991.296,E2 -20991.296} C_VEL
LIN {X 0,Y 375.501,Z 772.355,A -85,B 0,C 180,E1 -20992.05,E2 -20992.05} C_VEL
LIN {X 0,Y 377.136,Z 760.763,A -85,B 0,C 180,E1 -20992.668,E2 -20992.668} C_VEL
LIN {X 0,Y 378.228,Z 750.248,A -85,B 0,C 180,E1 -20993.103,E2 -20993.103} C_VEL
LIN {X 0,Y 382.589,Z 692.58,A -85,B 0,C 180,E1 -20994.829,E2 -20994.829} C_VEL
LIN {X 0,Y 380.956,Z 680.156,A -85,B 0,C 180,E1 -20995.55,E2 -20995.55} C_VEL
LIN {X 0,Y 378.343,Z 666.746,A -85,B 0,C 180,E1 -20996.48,E2 -20996.48} C_VEL
LIN {X 0,Y 376.834,Z 660.951,A -85,B 0,C 180,E1 -20996.964,E2 -20996.964} C_VEL
LIN {X 0,Y 371.984,Z 650.737,A -85,B 0,C 180,E1 -20998.2,E2 -20998.2} C_VEL
LIN {X 0,Y 369.572,Z 646.199,A -85,B 0,C 180,E1 -20998.839,E2 -20998.839} C_VEL
LIN {X 0,Y 366.66,Z 641.068,A -85,B 0,C 180,E1 -20999.631,E2 -20999.631} C_VEL
LIN {X 0,Y 366.364,Z 640.182,A -85,B 0,C 180,E1 -20999.808,E2 -20999.808} C_VEL
LIN {X 0,Y 365.028,Z 634.281,A -85,B 0,C 180,E1 -21002.499,E2 -21002.499} C_VEL
LIN {X 0,Y 363.774,Z 628.935,A -85,B 0,C 180,E1 -21005.286,E2 -21005.286} C_VEL
LIN {X 0,Y 362.509,Z 624.25,A -85,B 0,C 180,E1 -21008.193,E2 -21008.193} C_VEL
LIN {X 0,Y 361.277,Z 620.379,A -85,B 0,C 180,E1 -21011.239,E2 -21011.239} C_VEL
LIN {X 0,Y 360.357,Z 617.429,A -85,B 0,C 180,E1 -21014.407,E2 -21014.407} C_VEL
LIN {X 0,Y 359.802,Z 615.42,A -85,B 0,C 180,E1 -21017.712,E2 -21017.712} C_VEL
LIN {X 0,Y 359.486,Z 614.655,A -85,B 0,C 180,E1 -21021.205,E2 -21021.205} C_VEL
LIN {X 0,Y 359.725,Z 615.145,A -85,B 0,C 180,E1 -21024.867,E2 -21024.867} C_VEL
LIN {X 0,Y 360.371,Z 617.299,A -85,B 0,C 180,E1 -21028.784,E2 -21028.784} C_VEL
LIN {X 0,Y 361.346,Z 620.487,A -85,B 0,C 180,E1 -21032.275,E2 -21032.275} C_VEL
LIN {X 0,Y 362.381,Z 624.288,A -85,B 0,C 180,E1 -21035.294,E2 -21035.294} C_VEL
LIN {X 0,Y 363.72,Z 629.319,A -85,B 0,C 180,E1 -21038.537,E2 -21038.537} C_VEL
LIN {X 0,Y 364.45,Z 632.082,A -85,B 0,C 180,E1 -21039.983,E2 -21039.983} C_VEL
LIN {X 0,Y 366.776,Z 635.983,A -85,B 0,C 180,E1 -21040.637,E2 -21040.637} C_VEL
LIN {X 0,Y 368.092,Z 637.924,A -85,B 0,C 180,E1 -21040.982,E2 -21040.982} C_VEL
LIN {X 0,Y 371.379,Z 643.554,A -85,B 0,C 180,E1 -21041.862,E2 -21041.862} C_VEL
LIN {X 0,Y 375.477,Z 650.659,A -85,B 0,C 180,E1 -21042.865,E2 -21042.865} C_VEL
LIN {X 0,Y 380.792,Z 661.414,A -85,B 0,C 180,E1 -21044.15,E2 -21044.15} C_VEL
LIN {X 0,Y 382.706,Z 666.143,A -85,B 0,C 180,E1 -21044.61,E2 -21044.61} C_VEL
LIN {X 0,Y 383.85,Z 673.071,A -85,B 0,C 180,E1 -21045.046,E2 -21045.046} C_VEL
LIN {X 0,Y 378.697,Z 736.816,A -85,B 0,C 180,E1 -21046.938,E2 -21046.938} C_VEL
LIN {X 0,Y 377.686,Z 746.956,A -85,B 0,C 180,E1 -21047.345,E2 -21047.345} C_VEL
LIN {X 0,Y 376.511,Z 756.598,A -85,B 0,C 180,E1 -21047.851,E2 -21047.851} C_VEL
LIN {X 0,Y 375.019,Z 767.105,A -85,B 0,C 180,E1 -21048.553,E2 -21048.553} C_VEL
LIN {X 0,Y 373.484,Z 776.474,A -85,B 0,C 180,E1 -21049.327,E2 -21049.327} C_VEL
LIN {X 0,Y 371.746,Z 785.63,A -85,B 0,C 180,E1 -21050.236,E2 -21050.236} C_VEL
LIN {X 0,Y 369.937,Z 794.392,A -85,B 0,C 180,E1 -21051.287,E2 -21051.287} C_VEL
LIN {X 0,Y 368.192,Z 801.888,A -85,B 0,C 180,E1 -21052.347,E2 -21052.347} C_VEL
LIN {X 0,Y 366.16,Z 809.813,A -85,B 0,C 180,E1 -21053.685,E2 -21053.685} C_VEL
LIN {X 0,Y 364.292,Z 816.496,A -85,B 0,C 180,E1 -21055.036,E2 -21055.036} C_VEL
LIN {X 0,Y 362.929,Z 821.128,A -85,B 0,C 180,E1 -21056.126,E2 -21056.126} C_VEL
LIN {X 0,Y 361.149,Z 826.746,A -85,B 0,C 180,E1 -21057.777,E2 -21057.777} C_VEL
LIN {X 0,Y 359.682,Z 831.154,A -85,B 0,C 180,E1 -21059.442,E2 -21059.442} C_VEL
LIN {X 0,Y 358.54,Z 834.47,A -85,B 0,C 180,E1 -21061.119,E2 -21061.119} C_VEL
LIN {X 0,Y 357.703,Z 836.904,A -85,B 0,C 180,E1 -21062.95,E2 -21062.95} C_VEL
LIN {X 0,Y 357.075,Z 838.136,A -85,B 0,C 180,E1 -21064.5,E2 -21064.5} C_VEL
LIN {X 0,Y 356.448,Z 838.344,A -85,B 0,C 180,E1 -21066.771,E2 -21066.771} C_VEL
LIN {X 0,Y 356.289,Z 837.923,A -85,B 0,C 180,E1 -21067.91,E2 -21067.91} C_VEL
LIN {X 0,Y 356.254,Z 835.537,A -85,B 0,C 180,E1 -21070.192,E2 -21070.192} C_VEL
LIN {X 0,Y 356.193,Z 832.578,A -85,B 0,C 180,E1 -21071.916,E2 -21071.916} C_VEL
LIN {X 0,Y 356.295,Z 830.064,A -85,B 0,C 180,E1 -21073.066,E2 -21073.066} C_VEL
LIN {X 0,Y 356.543,Z 825.135,A -85,B 0,C 180,E1 -21074.796,E2 -21074.796} C_VEL
LIN {X 0,Y 356.86,Z 818.75,A -85,B 0,C 180,E1 -21076.535,E2 -21076.535} C_VEL
LIN {X 0,Y 357.166,Z 812.189,A -85,B 0,C 180,E1 -21077.991,E2 -21077.991} C_VEL
LIN {X 0,Y 357.646,Z 804.231,A -85,B 0,C 180,E1 -21079.447,E2 -21079.447} C_VEL
LIN {X 0,Y 358.143,Z 795.577,A -85,B 0,C 180,E1 -21080.761,E2 -21080.761} C_VEL
LIN {X 0,Y 358.606,Z 787.627,A -85,B 0,C 180,E1 -21081.784,E2 -21081.784} C_VEL
LIN {X 0,Y 359.179,Z 778.181,A -85,B 0,C 180,E1 -21082.804,E2 -21082.804} C_VEL
LIN {X 0,Y 359.766,Z 768.383,A -85,B 0,C 180,E1 -21083.681,E2 -21083.681} C_VEL
LIN {X 0,Y 360.29,Z 757.345,A -85,B 0,C 180,E1 -21084.477,E2 -21084.477} C_VEL
LIN {X 0,Y 360.605,Z 746.993,A -85,B 0,C 180,E1 -21085.067,E2 -21085.067} C_VEL
LIN {X 0,Y 361.024,Z 736.046,A -85,B 0,C 180,E1 -21085.536,E2 -21085.536} C_VEL
LIN {X 0,Y 361.806,Z 713.027,A -85,B 0,C 180,E1 -21086.208,E2 -21086.208} C_VEL
LIN {X 0,Y 363.183,Z 658.156,A -85,B 0,C 180,E1 -21087.74,E2 -21087.74} C_VEL
LIN {X 0,Y 360.116,Z 631.002,A -85,B 0,C 180,E1 -21088.579,E2 -21088.579} C_VEL
LIN {X 0,Y 359.866,Z 627.51,A -85,B 0,C 180,E1 -21088.696,E2 -21088.696} C_VEL
LIN {X 0,Y 360.417,Z 620.154,A -85,B 0,C 180,E1 -21090.741,E2 -21090.741} C_VEL
LIN {X 0,Y 359.094,Z 612.683,A -85,B 0,C 180,E1 -21092.946,E2 -21092.946} C_VEL
LIN {X 0,Y 358.956,Z 612.7,A -85,B 0,C 180,E1 -21097.222,E2 -21097.222} C_VEL
LIN {X 0,Y 358.929,Z 612.706,A -85,B 0,C 180,E1 -21100.44,E2 -21100.44} C_VEL
LIN {X 0,Y 358.98,Z 612.702,A -85,B 0,C 180,E1 -21103.784,E2 -21103.784} C_VEL
LIN {X 0,Y 358.973,Z 612.698,A -85,B 0,C 180,E1 -21106.926,E2 -21106.926} C_VEL
LIN {X 0,Y 358.913,Z 612.711,A -85,B 0,C 180,E1 -21109.908,E2 -21109.908} C_VEL
LIN {X 0,Y 358.962,Z 612.7,A -85,B 0,C 180,E1 -21113.132,E2 -21113.132} C_VEL
LIN {X 0,Y 358.953,Z 612.702,A -85,B 0,C 180,E1 -21115.535,E2 -21115.535} C_VEL
LIN {X 0,Y 359.001,Z 612.697,A -85,B 0,C 180,E1 -21119.517,E2 -21119.517} C_VEL
LIN {X 0,Y 358.966,Z 612.705,A -85,B 0,C 180,E1 -21122.075,E2 -21122.075} C_VEL
LIN {X 0,Y 358.966,Z 612.7,A -85,B 0,C 180,E1 -21124.578,E2 -21124.578} C_VEL
LIN {X 0,Y 358.98,Z 612.697,A -85,B 0,C 180,E1 -21127.03,E2 -21127.03} C_VEL
LIN {X 0,Y 359.012,Z 612.695,A -85,B 0,C 180,E1 -21130.629,E2 -21130.629} C_VEL
LIN {X 0,Y 359.062,Z 612.691,A -85,B 0,C 180,E1 -21134.151,E2 -21134.151} C_VEL
LIN {X 0,Y 359.159,Z 612.677,A -85,B 0,C 180,E1 -21137.612,E2 -21137.612} C_VEL
LIN {X 0,Y 359.186,Z 612.672,A -85,B 0,C 180,E1 -21141.025,E2 -21141.025} C_VEL
LIN {X 0,Y 359.298,Z 612.659,A -85,B 0,C 180,E1 -21144.406,E2 -21144.406} C_VEL
LIN {X 0,Y 359.331,Z 612.654,A -85,B 0,C 180,E1 -21146.647,E2 -21146.647} C_VEL
LIN {X 0,Y 359.331,Z 612.661,A -85,B 0,C 180,E1 -21150,E2 -21150} C_VEL
LIN {X 0,Y 359.33,Z 612.654,A -85,B 0,C 180,E1 -21153.352,E2 -21153.352} C_VEL
LIN {X 0,Y 359.294,Z 612.659,A -85,B 0,C 180,E1 -21156.717,E2 -21156.717} C_VEL
LIN {X 0,Y 359.138,Z 612.683,A -85,B 0,C 180,E1 -21160.109,E2 -21160.109} C_VEL
LIN {X 0,Y 359.096,Z 612.685,A -85,B 0,C 180,E1 -21163.537,E2 -21163.537} C_VEL
LIN {X 0,Y 359.085,Z 612.684,A -85,B 0,C 180,E1 -21167.099,E2 -21167.099} C_VEL
LIN {X 0,Y 359.024,Z 612.693,A -85,B 0,C 180,E1 -21170.559,E2 -21170.559} C_VEL
LIN {X 0,Y 358.96,Z 612.704,A -85,B 0,C 180,E1 -21174.191,E2 -21174.191} C_VEL
LIN {X 0,Y 358.954,Z 612.701,A -85,B 0,C 180,E1 -21176.667,E2 -21176.667} C_VEL
LIN {X 0,Y 358.957,Z 612.701,A -85,B 0,C 180,E1 -21179.198,E2 -21179.198} C_VEL
LIN {X 0,Y 358.962,Z 612.704,A -85,B 0,C 180,E1 -21181.793,E2 -21181.793} C_VEL
LIN {X 0,Y 359.03,Z 612.695,A -85,B 0,C 180,E1 -21185.823,E2 -21185.823} C_VEL
LIN {X 0,Y 358.989,Z 612.697,A -85,B 0,C 180,E1 -21188.698,E2 -21188.698} C_VEL
LIN {X 0,Y 358.946,Z 612.706,A -85,B 0,C 180,E1 -21192.139,E2 -21192.139} C_VEL
LIN {X 0,Y 358.966,Z 612.7,A -85,B 0,C 180,E1 -21195.376,E2 -21195.376} C_VEL
LIN {X 0,Y 358.955,Z 612.703,A -85,B 0,C 180,E1 -21198.437,E2 -21198.437} C_VEL
LIN {X 0,Y 358.957,Z 612.701,A -85,B 0,C 180,E1 -21201.361,E2 -21201.361} C_VEL
LIN {X 0,Y 358.964,Z 612.699,A -85,B 0,C 180,E1 -21205.039,E2 -21205.039} C_VEL
LIN {X 0,Y 358.973,Z 612.699,A -85,B 0,C 180,E1 -21209.154,E2 -21209.154} C_VEL
LIN {X 0,Y 358.966,Z 612.704,A -85,B 0,C 180,E1 -21212.076,E2 -21212.076} C_VEL
LIN {X 0,Y 358.967,Z 612.7,A -85,B 0,C 180,E1 -21214.579,E2 -21214.579} C_VEL
LIN {X 0,Y 358.982,Z 612.697,A -85,B 0,C 180,E1 -21217.031,E2 -21217.031} C_VEL
LIN {X 0,Y 359.009,Z 612.695,A -85,B 0,C 180,E1 -21220.63,E2 -21220.63} C_VEL
LIN {X 0,Y 359.011,Z 612.698,A -85,B 0,C 180,E1 -21224.149,E2 -21224.149} C_VEL
LIN {X 0,Y 359.156,Z 612.678,A -85,B 0,C 180,E1 -21227.613,E2 -21227.613} C_VEL
LIN {X 0,Y 359.191,Z 612.671,A -85,B 0,C 180,E1 -21231.025,E2 -21231.025} C_VEL
LIN {X 0,Y 359.414,Z 612.645,A -85,B 0,C 180,E1 -21233.674,E2 -21233.674} C_VEL
LIN {X 0,Y 359.334,Z 612.654,A -85,B 0,C 180,E1 -21236.648,E2 -21236.648} C_VEL
LIN {X 0,Y 359.333,Z 612.66,A -85,B 0,C 180,E1 -21240,E2 -21240} C_VEL
LIN {X 0,Y 359.318,Z 612.654,A -85,B 0,C 180,E1 -21243.036,E2 -21243.036} C_VEL
LIN {X 0,Y 358.674,Z 612.741,A -85,B 0,C 180,E1 -21243.972,E2 -21243.972} C_VEL
LIN {X 0,Y 355.826,Z 613.103,A -85,B 0,C 180,E1 -21245.495,E2 -21245.495} C_VEL
LIN {X 0,Y 353.375,Z 613.411,A -85,B 0,C 180,E1 -21246.727,E2 -21246.727} C_VEL
LIN {X 0,Y 352.288,Z 613.542,A -85,B 0,C 180,E1 -21247.68,E2 -21247.68} C_VEL
LIN {X 0,Y 352.181,Z 613.551,A -85,B 0,C 180,E1 -21248.003,E2 -21248.003} C_VEL
LIN {X 0,Y 352.091,Z 613.556,A -85,B 0,C 180,E1 -21251.475,E2 -21251.475} C_VEL
LIN {X 0,Y 352.007,Z 613.57,A -85,B 0,C 180,E1 -21253.815,E2 -21253.815} C_VEL
LIN {X 0,Y 351.944,Z 613.575,A -85,B 0,C 180,E1 -21257.37,E2 -21257.37} C_VEL
LIN {X 0,Y 351.903,Z 613.578,A -85,B 0,C 180,E1 -21260.995,E2 -21260.995} C_VEL
LIN {X 0,Y 351.944,Z 613.577,A -85,B 0,C 180,E1 -21263.724,E2 -21263.724} C_VEL
LIN {X 0,Y 351.911,Z 613.579,A -85,B 0,C 180,E1 -21267.245,E2 -21267.245} C_VEL
LIN {X 0,Y 351.895,Z 613.585,A -85,B 0,C 180,E1 -21269.843,E2 -21269.843} C_VEL
LIN {X 0,Y 351.878,Z 613.587,A -85,B 0,C 180,E1 -21273.874,E2 -21273.874} C_VEL
LIN {X 0,Y 351.903,Z 613.58,A -85,B 0,C 180,E1 -21277.233,E2 -21277.233} C_VEL
LIN {X 0,Y 351.859,Z 613.583,A -85,B 0,C 180,E1 -21281.066,E2 -21281.066} C_VEL
LIN {X 0,Y 351.871,Z 613.587,A -85,B 0,C 180,E1 -21284.224,E2 -21284.224} C_VEL
LIN {X 0,Y 351.871,Z 613.585,A -85,B 0,C 180,E1 -21287.437,E2 -21287.437} C_VEL
LIN {X 0,Y 351.857,Z 613.583,A -85,B 0,C 180,E1 -21290.93,E2 -21290.93} C_VEL
LIN {X 0,Y 351.883,Z 613.582,A -85,B 0,C 180,E1 -21293.333,E2 -21293.333} C_VEL
LIN {X 0,Y 351.862,Z 613.585,A -85,B 0,C 180,E1 -21296.729,E2 -21296.729} C_VEL
LIN {X 0,Y 351.882,Z 613.585,A -85,B 0,C 180,E1 -21300.156,E2 -21300.156} C_VEL
LIN {X 0,Y 352.01,Z 613.591,A -85,B 0,C 180,E1 -21303.184,E2 -21303.184} C_VEL
LIN {X 0,Y 354.219,Z 626.434,A -85,B 0,C 180,E1 -21306.704,E2 -21306.704} C_VEL
LIN {X 0,Y 353.912,Z 631.048,A -85,B 0,C 180,E1 -21307.912,E2 -21307.912} C_VEL
LIN {X 0,Y 352.448,Z 643.413,A -85,B 0,C 180,E1 -21311.121,E2 -21311.121} C_VEL
LIN {X 0,Y 354.137,Z 667.378,A -85,B 0,C 180,E1 -21311.888,E2 -21311.888} C_VEL
LIN {X 0,Y 355.821,Z 685.127,A -85,B 0,C 180,E1 -21312.439,E2 -21312.439} C_VEL
LIN {X 0,Y 354.071,Z 750.293,A -85,B 0,C 180,E1 -21314.327,E2 -21314.327} C_VEL
LIN {X 0,Y 353.637,Z 760.589,A -85,B 0,C 180,E1 -21314.748,E2 -21314.748} C_VEL
LIN {X 0,Y 353.301,Z 770.453,A -85,B 0,C 180,E1 -21315.285,E2 -21315.285} C_VEL
LIN {X 0,Y 352.849,Z 779.877,A -85,B 0,C 180,E1 -21315.926,E2 -21315.926} C_VEL
LIN {X 0,Y 352.299,Z 790.657,A -85,B 0,C 180,E1 -21316.841,E2 -21316.841} C_VEL
LIN {X 0,Y 351.616,Z 799.682,A -85,B 0,C 180,E1 -21317.771,E2 -21317.771} C_VEL
LIN {X 0,Y 351.146,Z 808.001,A -85,B 0,C 180,E1 -21318.785,E2 -21318.785} C_VEL
LIN {X 0,Y 350.646,Z 815.975,A -85,B 0,C 180,E1 -21319.934,E2 -21319.934} C_VEL
LIN {X 0,Y 350.139,Z 824.277,A -85,B 0,C 180,E1 -21321.371,E2 -21321.371} C_VEL
LIN {X 0,Y 349.861,Z 831.2,A -85,B 0,C 180,E1 -21322.812,E2 -21322.812} C_VEL
LIN {X 0,Y 349.652,Z 836.951,A -85,B 0,C 180,E1 -21324.252,E2 -21324.252} C_VEL
LIN {X 0,Y 349.544,Z 840.87,A -85,B 0,C 180,E1 -21325.403,E2 -21325.403} C_VEL
LIN {X 0,Y 349.497,Z 845.545,A -85,B 0,C 180,E1 -21327.128,E2 -21327.128} C_VEL
LIN {X 0,Y 349.434,Z 849.042,A -85,B 0,C 180,E1 -21328.852,E2 -21328.852} C_VEL
LIN {X 0,Y 349.366,Z 851.97,A -85,B 0,C 180,E1 -21331.149,E2 -21331.149} C_VEL
LIN {X 0,Y 349.332,Z 852.9,A -85,B 0,C 180,E1 -21332.299,E2 -21332.299} C_VEL
LIN {X 0,Y 349.379,Z 853.258,A -85,B 0,C 180,E1 -21334.6,E2 -21334.6} C_VEL
LIN {X 0,Y 349.57,Z 852.85,A -85,B 0,C 180,E1 -21335.75,E2 -21335.75} C_VEL
LIN {X 0,Y 350.228,Z 850.776,A -85,B 0,C 180,E1 -21338.048,E2 -21338.048} C_VEL
LIN {X 0,Y 351.112,Z 848.101,A -85,B 0,C 180,E1 -21339.763,E2 -21339.763} C_VEL
LIN {X 0,Y 352.223,Z 844.399,A -85,B 0,C 180,E1 -21341.471,E2 -21341.471} C_VEL
LIN {X 0,Y 353.809,Z 839.566,A -85,B 0,C 180,E1 -21343.16,E2 -21343.16} C_VEL
LIN {X 0,Y 355.707,Z 833.463,A -85,B 0,C 180,E1 -21344.833,E2 -21344.833} C_VEL
LIN {X 0,Y 357.646,Z 826.26,A -85,B 0,C 180,E1 -21346.44,E2 -21346.44} C_VEL
LIN {X 0,Y 359.888,Z 818.45,A -85,B 0,C 180,E1 -21347.851,E2 -21347.851} C_VEL
LIN {X 0,Y 361.686,Z 811.456,A -85,B 0,C 180,E1 -21348.928,E2 -21348.928} C_VEL
LIN {X 0,Y 363.895,Z 802.084,A -85,B 0,C 180,E1 -21350.125,E2 -21350.125} C_VEL
LIN {X 0,Y 366.047,Z 792.07,A -85,B 0,C 180,E1 -21351.173,E2 -21351.173} C_VEL
LIN {X 0,Y 368.146,Z 781.397,A -85,B 0,C 180,E1 -21352.072,E2 -21352.072} C_VEL
LIN {X 0,Y 370.129,Z 770.134,A -85,B 0,C 180,E1 -21352.827,E2 -21352.827} C_VEL
LIN {X 0,Y 371.642,Z 759.566,A -85,B 0,C 180,E1 -21353.389,E2 -21353.389} C_VEL
LIN {X 0,Y 372.839,Z 748.89,A -85,B 0,C 180,E1 -21353.823,E2 -21353.823} C_VEL
LIN {X 0,Y 377.174,Z 693.595,A -85,B 0,C 180,E1 -21355.513,E2 -21355.513} C_VEL
LIN {X 0,Y 375.324,Z 680.03,A -85,B 0,C 180,E1 -21356.352,E2 -21356.352} C_VEL
LIN {X 0,Y 372.622,Z 666.132,A -85,B 0,C 180,E1 -21357.396,E2 -21357.396} C_VEL
LIN {X 0,Y 369.183,Z 658.574,A -85,B 0,C 180,E1 -21358.301,E2 -21358.301} C_VEL
LIN {X 0,Y 364.864,Z 650.064,A -85,B 0,C 180,E1 -21359.511,E2 -21359.511} C_VEL
